C09144=1176.227,126.647,-53.704,-178.669,6.349,148.760
C09145=1176.232,126.397,-53.684,-178.672,6.347,148.760
C09146=1176.237,126.148,-53.664,-178.674,6.346,148.761
C09147=1176.242,125.899,-53.644,-178.677,6.344,148.761
C09148=1176.246,125.650,-53.625,-178.680,6.343,148.762
C09149=1176.251,125.401,-53.606,-178.683,6.341,148.762
C09150=1176.255,125.151,-53.586,-178.685,6.339,148.763
C09151=1176.260,124.903,-53.566,-178.688,6.338,148.763
C09152=1176.265,124.653,-53.546,-178.690,6.337,148.763
C09153=1176.270,124.404,-53.527,-178.693,6.335,148.764
C09154=1176.275,124.155,-53.507,-178.696,6.334,148.764
C09155=1176.280,123.906,-53.487,-178.698,6.333,148.765
C09156=1176.284,123.656,-53.467,-178.701,6.331,148.765
C09157=1176.290,123.407,-53.448,-178.704,6.330,148.766
C09158=1176.294,123.158,-53.429,-178.707,6.328,148.766
C09159=1176.299,122.909,-53.409,-178.709,6.327,148.767
C09160=1176.304,122.660,-53.390,-178.712,6.325,148.767
C09161=1176.308,122.411,-53.370,-178.715,6.324,148.768
C09162=1176.313,122.161,-53.350,-178.718,6.322,148.768
C09163=1176.318,121.912,-53.331,-178.720,6.321,148.768
C09164=1176.322,121.663,-53.312,-178.722,6.319,148.769
C09165=1176.327,121.414,-53.292,-178.726,6.318,148.769
C09166=1176.332,121.165,-53.273,-178.728,6.317,148.770
C09167=1176.337,120.915,-53.253,-178.730,6.315,148.770
C09168=1176.343,120.666,-53.234,-178.733,6.314,148.771
C09169=1176.347,120.417,-53.215,-178.736,6.312,148.771
C09170=1176.351,120.167,-53.195,-178.738,6.311,148.772
C09171=1176.357,119.919,-53.176,-178.741,6.310,148.772
C09172=1176.361,119.669,-53.156,-178.744,6.308,148.772
C09173=1176.366,119.420,-53.137,-178.747,6.306,148.773
C09174=1176.371,119.171,-53.118,-178.749,6.306,148.774
C09175=1176.375,118.921,-53.098,-178.752,6.304,148.774
C09176=1176.381,118.672,-53.079,-178.755,6.302,148.774
C09177=1176.385,118.423,-53.060,-178.757,6.302,148.775
C09178=1176.390,118.174,-53.041,-178.760,6.300,148.775
C09179=1176.395,117.925,-53.021,-178.763,6.298,148.776
C09180=1176.400,117.676,-53.002,-178.766,6.297,148.776
C09181=1176.404,117.427,-52.983,-178.768,6.296,148.777
C09182=1176.409,117.177,-52.963,-178.771,6.294,148.777
C09183=1176.414,116.928,-52.944,-178.773,6.292,148.778
C09184=1176.418,116.679,-52.925,-178.776,6.292,148.778
C09185=1176.424,116.430,-52.905,-178.779,6.290,148.779
C09186=1176.428,116.180,-52.886,-178.781,6.288,148.779
C09187=1176.433,115.931,-52.868,-178.783,6.287,148.779
C09188=1176.438,115.682,-52.848,-178.787,6.286,148.780
C09189=1176.443,115.433,-52.829,-178.789,6.284,148.780
C09190=1176.447,115.184,-52.810,-178.792,6.283,148.781
C09191=1176.453,114.935,-52.790,-178.795,6.282,148.782
C09192=1176.458,114.685,-52.771,-178.797,6.280,148.782
C09193=1176.462,114.436,-52.753,-178.800,6.278,148.782
C09194=1176.467,114.186,-52.733,-178.802,6.278,148.783
C09195=1176.473,113.938,-52.714,-178.805,6.276,148.783
C09196=1176.477,113.688,-52.695,-178.808,6.274,148.784
C09197=1176.482,113.439,-52.675,-178.810,6.274,148.784
C09198=1176.486,113.190,-52.657,-178.813,6.272,148.785
C09199=1176.492,112.941,-52.638,-178.816,6.270,148.785
C09200=1176.496,112.691,-52.619,-178.818,6.270,148.786
C09201=1176.501,112.443,-52.599,-178.822,6.268,148.786
C09202=1176.506,112.192,-52.580,-178.824,6.266,148.787
C09203=1176.511,111.944,-52.562,-178.826,6.266,148.787
C09204=1176.515,111.694,-52.542,-178.829,6.264,148.787
C09205=1176.520,111.445,-52.524,-178.832,6.262,148.788
C09206=1176.526,111.196,-52.505,-178.834,6.261,148.789
C09207=1176.530,110.947,-52.486,-178.837,6.260,148.789
C09208=1176.535,110.697,-52.467,-178.840,6.258,148.790
C09209=1176.539,110.448,-52.448,-178.842,6.257,148.790
C09210=1176.545,110.199,-52.429,-178.845,6.256,148.790
C09211=1176.549,109.949,-52.410,-178.848,6.254,148.791
C09212=1176.554,109.701,-52.391,-178.850,6.253,148.791
C09213=1176.559,109.451,-52.373,-178.853,6.252,148.792
C09214=1176.564,109.202,-52.354,-178.856,6.250,148.792
C09215=1176.568,108.953,-52.335,-178.859,6.249,148.793
C09216=1176.574,108.703,-52.316,-178.861,6.248,148.793
C09217=1176.578,108.455,-52.297,-178.864,6.246,148.794
C09218=1176.584,108.205,-52.279,-178.867,6.245,148.794
C09219=1176.588,107.956,-52.260,-178.869,6.244,148.795
C09220=1176.593,107.707,-52.242,-178.872,6.242,148.795
C09221=1176.597,107.457,-52.222,-178.875,6.241,148.796
C09222=1176.602,107.208,-52.204,-178.877,6.240,148.796
C09223=1176.608,106.959,-52.185,-178.880,6.239,148.797
C09224=1176.612,106.690,-52.165,-178.883,6.237,148.797
C09225=1176.618,106.422,-52.144,-178.886,6.236,148.798
C09226=1176.623,106.154,-52.125,-178.889,6.234,148.798
C09227=1176.628,105.885,-52.104,-178.892,6.233,148.799
C09228=1176.633,105.636,-52.086,-178.894,6.232,148.799
C09229=1176.638,105.387,-52.067,-178.897,6.230,148.800
C09230=1176.642,105.137,-52.048,-178.900,6.229,148.800
C09231=1176.647,104.888,-52.030,-178.902,6.228,148.801
C09232=1176.653,104.639,-52.011,-178.905,6.226,148.801
C09233=1176.657,104.389,-51.992,-178.908,6.225,148.802
C09234=1176.662,104.140,-51.974,-178.910,6.224,148.802
C09235=1176.667,103.891,-51.955,-178.913,6.222,148.803
C09236=1176.671,103.641,-51.937,-178.915,6.222,148.803
C09237=1176.676,103.392,-51.919,-178.918,6.220,148.804
C09238=1176.682,103.143,-51.900,-178.921,6.218,148.804
C09239=1176.687,102.894,-51.882,-178.923,6.218,148.805
C09240=1176.691,102.644,-51.863,-178.926,6.216,148.805
C09241=1176.695,102.396,-51.845,-178.928,6.215,148.806
C09242=1176.701,102.146,-51.826,-178.931,6.214,148.806
C09243=1176.705,101.896,-51.808,-178.934,6.212,148.807
C09244=1176.710,101.648,-51.789,-178.937,6.212,148.807
C09245=1176.716,101.398,-51.770,-178.939,6.210,148.808
C09246=1176.721,101.149,-51.752,-178.942,6.209,148.808
C09247=1176.725,100.899,-51.734,-178.945,6.208,148.809
C09248=1176.730,100.651,-51.715,-178.947,6.206,148.809
C09249=1176.735,100.401,-51.697,-178.950,6.205,148.810
C09250=1176.740,100.152,-51.679,-178.953,6.204,148.810
C09251=1176.744,99.902,-51.660,-178.955,6.203,148.811
C09252=1176.749,99.654,-51.642,-178.958,6.201,148.811
C09253=1176.754,99.405,-51.624,-178.961,6.200,148.812
C09254=1176.760,99.155,-51.605,-178.963,6.199,148.812
C09255=1176.764,98.905,-51.587,-178.966,6.197,148.813
C09256=1176.769,98.656,-51.569,-178.968,6.196,148.813
C09257=1176.773,98.407,-51.550,-178.971,6.195,148.814
C09258=1176.778,98.158,-51.532,-178.974,6.193,148.814
C09259=1176.783,97.909,-51.514,-178.976,6.192,148.815
C09260=1176.788,97.659,-51.495,-178.979,6.191,148.815
C09261=1176.793,97.410,-51.477,-178.982,6.190,148.816
C09262=1176.798,97.161,-51.459,-178.984,6.188,148.816
C09263=1176.803,96.911,-51.441,-178.987,6.188,148.817
C09264=1176.808,96.662,-51.423,-178.990,6.186,148.817
C09265=1176.812,96.412,-51.405,-178.992,6.184,148.818
C09266=1176.817,96.164,-51.386,-178.995,6.184,148.818
C09267=1176.822,95.915,-51.368,-178.998,6.182,148.819
C09268=1176.827,95.665,-51.350,-179.000,6.182,148.819
C09269=1176.832,95.416,-51.332,-179.003,6.180,148.820
C09270=1176.837,95.167,-51.314,-179.005,6.179,148.820
C09271=1176.842,94.917,-51.295,-179.008,6.178,148.821
C09272=1176.846,94.668,-51.277,-179.011,6.177,148.821
C09273=1176.851,94.419,-51.259,-179.014,6.175,148.822
C09274=1176.856,94.169,-51.241,-179.017,6.174,148.822
C09275=1176.861,93.920,-51.224,-179.019,6.173,148.823
C09276=1176.866,93.671,-51.206,-179.022,6.171,148.823
C09277=1176.871,93.422,-51.188,-179.024,6.171,148.824
C09278=1176.875,93.172,-51.169,-179.027,6.169,148.824
C09279=1176.880,92.923,-51.151,-179.029,6.168,148.825
C09280=1176.885,92.673,-51.134,-179.032,6.167,148.825
C09281=1176.890,92.424,-51.116,-179.035,6.166,148.826
C09282=1176.895,92.175,-51.098,-179.037,6.164,148.826
C09283=1176.900,91.925,-51.080,-179.041,6.163,148.827
C09284=1176.905,91.676,-51.062,-179.043,6.162,148.827
C09285=1176.910,91.427,-51.044,-179.045,6.160,148.828
C09286=1176.915,91.178,-51.026,-179.048,6.160,148.828
C09287=1176.920,90.929,-51.008,-179.051,6.158,148.829
C09288=1176.924,90.679,-50.990,-179.053,6.158,148.829
C09289=1176.929,90.429,-50.972,-179.056,6.156,148.830
C09290=1176.934,90.180,-50.955,-179.058,6.155,148.830
C09291=1176.939,89.931,-50.937,-179.062,6.154,148.831
C09292=1176.944,89.682,-50.919,-179.064,6.153,148.831
C09293=1176.949,89.432,-50.901,-179.067,6.151,148.832
C09294=1176.954,89.183,-50.883,-179.069,6.150,148.832
C09295=1176.959,88.933,-50.865,-179.072,6.149,148.833
C09296=1176.963,88.685,-50.848,-179.074,6.148,148.833
C09297=1176.968,88.435,-50.830,-179.077,6.146,148.834
C09298=1176.973,88.186,-50.812,-179.080,6.146,148.835
C09299=1176.978,87.936,-50.795,-179.082,6.144,148.835
C09300=1176.983,87.687,-50.777,-179.085,6.144,148.836
C09301=1176.988,87.438,-50.759,-179.088,6.142,148.836
C09302=1176.993,87.188,-50.741,-179.090,6.141,148.837
C09303=1176.998,86.939,-50.724,-179.093,6.140,148.837
C09304=1177.003,86.690,-50.706,-179.095,6.139,148.838
C09305=1177.007,86.441,-50.688,-179.098,6.137,148.838
C09306=1177.013,86.191,-50.671,-179.101,6.137,148.839
C09307=1177.018,85.942,-50.653,-179.104,6.135,148.839
C09308=1177.022,85.693,-50.635,-179.106,6.134,148.840
C09309=1177.028,85.443,-50.618,-179.109,6.133,148.840
C09310=1177.032,85.194,-50.600,-179.111,6.132,148.841
C09311=1177.037,84.944,-50.583,-179.114,6.130,148.841
C09312=1177.042,84.695,-50.565,-179.117,6.130,148.842
C09313=1177.047,84.446,-50.547,-179.119,6.128,148.842
C09314=1177.052,84.196,-50.530,-179.122,6.128,148.843
C09315=1177.056,83.947,-50.512,-179.125,6.126,148.843
C09316=1177.061,83.698,-50.495,-179.127,6.125,148.844
C09317=1177.066,83.448,-50.477,-179.130,6.124,148.844
C09318=1177.071,83.199,-50.459,-179.133,6.123,148.845
C09319=1177.077,82.949,-50.442,-179.135,6.121,148.845
C09320=1177.081,82.701,-50.425,-179.138,6.120,148.846
C09321=1177.086,82.451,-50.407,-179.141,6.119,148.847
C09322=1177.091,82.202,-50.389,-179.143,6.118,148.847
C09323=1177.095,81.952,-50.373,-179.146,6.117,148.848
C09324=1177.100,81.703,-50.355,-179.148,6.116,148.848
C09325=1177.106,81.454,-50.338,-179.151,6.115,148.849
C09326=1177.111,81.205,-50.320,-179.154,6.114,148.849
C09327=1177.115,80.955,-50.303,-179.157,6.112,148.850
C09328=1177.120,80.687,-50.284,-179.159,6.111,148.850
C09329=1177.126,80.418,-50.265,-179.162,6.110,148.851
C09330=1177.132,80.150,-50.247,-179.165,6.109,148.852
C09331=1177.137,79.881,-50.229,-179.167,6.108,148.852
C09332=1177.141,79.632,-50.211,-179.171,6.107,148.853
C09333=1177.147,79.382,-50.193,-179.173,6.106,148.853
C09334=1177.151,79.134,-50.176,-179.176,6.104,148.854
C09335=1177.156,78.884,-50.159,-179.178,6.103,148.854
C09336=1177.161,78.634,-50.141,-179.181,6.103,148.855
C09337=1177.166,78.386,-50.124,-179.184,6.101,148.855
C09338=1177.171,78.136,-50.107,-179.186,6.101,148.856
C09339=1177.175,77.887,-50.090,-179.189,6.099,148.856
C09340=1177.181,77.637,-50.072,-179.191,6.098,148.857
C09341=1177.186,77.388,-50.055,-179.194,6.097,148.857
C09342=1177.190,77.139,-50.038,-179.196,6.096,148.858
C09343=1177.195,76.889,-50.021,-179.200,6.094,148.858
C09344=1177.200,76.640,-50.004,-179.202,6.094,148.859
C09345=1177.205,76.391,-49.986,-179.204,6.093,148.860
C09346=1177.210,76.141,-49.969,-179.207,6.091,148.860
C09347=1177.215,75.892,-49.952,-179.210,6.091,148.861
C09348=1177.220,75.642,-49.935,-179.212,6.089,148.861
C09349=1177.225,75.394,-49.918,-179.215,6.089,148.862
C09350=1177.230,75.144,-49.901,-179.218,6.087,148.862
C09351=1177.235,74.894,-49.884,-179.220,6.086,148.863
C09352=1177.240,74.645,-49.867,-179.223,6.085,148.863
C09353=1177.244,74.396,-49.849,-179.226,6.084,148.864
C09354=1177.250,74.147,-49.833,-179.228,6.083,148.864
C09355=1177.254,73.897,-49.816,-179.231,6.082,148.865
C09356=1177.260,73.647,-49.799,-179.233,6.081,148.865
C09357=1177.264,73.398,-49.782,-179.237,6.080,148.866
C09358=1177.269,73.149,-49.764,-179.239,6.079,148.866
C09359=1177.274,72.900,-49.748,-179.241,6.078,148.867
C09360=1177.279,72.650,-49.730,-179.244,6.077,148.868
C09361=1177.284,72.401,-49.714,-179.247,6.076,148.868
C09362=1177.289,72.151,-49.696,-179.249,6.074,148.869
C09363=1177.294,71.902,-49.680,-179.252,6.074,148.869
C09364=1177.299,71.652,-49.663,-179.255,6.072,148.870
C09365=1177.304,71.403,-49.646,-179.257,6.072,148.870
C09366=1177.309,71.154,-49.628,-179.260,6.071,148.871
C09367=1177.314,70.905,-49.612,-179.263,6.069,148.871
C09368=1177.319,70.655,-49.595,-179.265,6.068,148.872
C09369=1177.323,70.406,-49.578,-179.268,6.067,148.873
C09370=1177.328,70.156,-49.561,-179.270,6.066,148.873
C09371=1177.334,69.907,-49.544,-179.273,6.066,148.874
C09372=1177.338,69.657,-49.528,-179.276,6.064,148.874
C09373=1177.343,69.408,-49.511,-179.278,6.063,148.875
C09374=1177.348,69.159,-49.494,-179.281,6.062,148.875
C09375=1177.353,68.909,-49.478,-179.284,6.061,148.876
C09376=1177.358,68.660,-49.460,-179.286,6.060,148.876
C09377=1177.363,68.410,-49.444,-179.289,6.059,148.877
C09378=1177.368,68.161,-49.427,-179.291,6.058,148.877
C09379=1177.373,67.912,-49.410,-179.294,6.058,148.878
C09380=1177.377,67.662,-49.393,-179.296,6.056,148.878
C09381=1177.383,67.413,-49.377,-179.299,6.055,148.879
C09382=1177.388,67.163,-49.360,-179.302,6.054,148.880
C09383=1177.392,66.914,-49.343,-179.304,6.053,148.880
C09384=1177.397,66.665,-49.327,-179.307,6.052,148.881
C09385=1177.403,66.415,-49.310,-179.310,6.051,148.881
C09386=1177.407,66.166,-49.293,-179.312,6.050,148.882
C09387=1177.412,65.917,-49.277,-179.315,6.050,148.882
C09388=1177.418,65.667,-49.260,-179.317,6.048,148.883
C09389=1177.422,65.417,-49.243,-179.320,6.047,148.883
C09390=1177.427,65.168,-49.227,-179.323,6.046,148.884
C09391=1177.432,64.919,-49.210,-179.325,6.045,148.885
C09392=1177.437,64.669,-49.193,-179.327,6.044,148.885
C09393=1177.442,64.420,-49.177,-179.331,6.043,148.886
C09394=1177.446,64.171,-49.160,-179.333,6.042,148.886
C09395=1177.452,63.922,-49.145,-179.335,6.042,148.887
C09396=1177.457,63.672,-49.127,-179.339,6.040,148.887
C09397=1177.462,63.422,-49.111,-179.341,6.039,148.888
C09398=1177.467,63.173,-49.094,-179.343,6.039,148.888
C09399=1177.471,62.924,-49.078,-179.346,6.037,148.889
C09400=1177.477,62.674,-49.062,-179.349,6.037,148.890
C09401=1177.482,62.425,-49.045,-179.352,6.035,148.890
C09402=1177.486,62.175,-49.028,-179.354,6.034,148.891
C09403=1177.491,61.927,-49.012,-179.356,6.033,148.891
C09404=1177.496,61.676,-48.996,-179.360,6.032,148.892
C09405=1177.502,61.427,-48.979,-179.362,6.031,148.892
C09406=1177.506,61.178,-48.962,-179.364,6.031,148.893
C09407=1177.511,60.929,-48.946,-179.367,6.029,148.893
C09408=1177.516,60.679,-48.930,-179.370,6.029,148.894
C09409=1177.521,60.429,-48.913,-179.372,6.028,148.895
C09410=1177.526,60.181,-48.897,-179.375,6.026,148.895
C09411=1177.531,59.930,-48.881,-179.378,6.026,148.896
C09412=1177.536,59.681,-48.864,-179.380,6.025,148.896
C09413=1177.541,59.432,-48.848,-179.383,6.024,148.897
C09414=1177.546,59.183,-48.832,-179.385,6.023,148.897
C09415=1177.551,58.933,-48.815,-179.388,6.022,148.898
C09416=1177.556,58.684,-48.799,-179.391,6.021,148.898
C09417=1177.561,58.434,-48.783,-179.393,6.020,148.899
C09418=1177.566,58.185,-48.767,-179.395,6.019,148.899
C09419=1177.571,57.935,-48.750,-179.399,6.018,148.900
C09420=1177.576,57.686,-48.734,-179.401,6.017,148.901
C09421=1177.581,57.437,-48.717,-179.403,6.016,148.901
C09422=1177.586,57.187,-48.702,-179.407,6.015,148.902
C09423=1177.591,56.938,-48.685,-179.409,6.014,148.902
C09424=1177.596,56.688,-48.669,-179.411,6.014,148.903
C09425=1177.600,56.439,-48.653,-179.414,6.013,148.903
C09426=1177.606,56.190,-48.637,-179.417,6.011,148.904
C09427=1177.610,55.940,-48.620,-179.419,6.011,148.905
C09428=1177.616,55.691,-48.605,-179.422,6.010,148.905
C09429=1177.620,55.441,-48.588,-179.425,6.009,148.906
C09430=1177.626,55.192,-48.573,-179.427,6.008,148.906
C09431=1177.630,54.942,-48.556,-179.430,6.007,148.907
C09432=1177.636,54.674,-48.539,-179.432,6.006,148.907
C09433=1177.641,54.405,-48.522,-179.435,6.005,148.908
C09434=1177.646,54.137,-48.504,-179.438,6.004,148.909
C09435=1177.651,53.868,-48.487,-179.441,6.003,148.909
C09436=1177.657,53.619,-48.471,-179.444,6.002,148.910
C09437=1177.661,53.369,-48.455,-179.446,6.001,148.911
C09438=1177.667,53.120,-48.439,-179.448,6.000,148.911
C09439=1177.671,52.870,-48.423,-179.451,6.000,148.912
C09440=1177.677,52.621,-48.407,-179.454,5.998,148.912
C09441=1177.682,52.372,-48.391,-179.456,5.998,148.913
C09442=1177.686,52.122,-48.374,-179.459,5.997,148.913
C09443=1177.692,51.873,-48.359,-179.462,5.995,148.914
C09444=1177.697,51.623,-48.343,-179.464,5.995,148.915
C09445=1177.702,51.374,-48.327,-179.466,5.994,148.915
C09446=1177.706,51.124,-48.311,-179.469,5.993,148.916
C09447=1177.712,50.875,-48.294,-179.472,5.992,148.916
C09448=1177.717,50.626,-48.279,-179.474,5.991,148.917
C09449=1177.722,50.376,-48.263,-179.477,5.991,148.917
C09450=1177.727,50.126,-48.247,-179.480,5.989,148.918
C09451=1177.731,49.877,-48.231,-179.483,5.989,148.919
C09452=1177.736,49.628,-48.216,-179.485,5.988,148.919
C09453=1177.742,49.378,-48.200,-179.487,5.987,148.920
C09454=1177.746,49.129,-48.183,-179.491,5.986,148.920
C09455=1177.751,48.879,-48.168,-179.493,5.985,148.921
C09456=1177.757,48.630,-48.152,-179.495,5.985,148.921
C09457=1177.762,48.380,-48.136,-179.497,5.984,148.922
C09458=1177.766,48.131,-48.120,-179.501,5.982,148.923
C09459=1177.771,47.882,-48.105,-179.503,5.981,148.923
C09460=1177.776,47.632,-48.089,-179.505,5.981,148.924
C09461=1177.782,47.382,-48.073,-179.508,5.980,148.924
C09462=1177.787,47.134,-48.057,-179.511,5.979,148.925
C09463=1177.791,46.884,-48.041,-179.514,5.978,148.925
C09464=1177.796,46.634,-48.026,-179.516,5.977,148.926
C09465=1177.801,46.385,-48.011,-179.518,5.977,148.927
C09466=1177.806,46.135,-47.995,-179.522,5.976,148.927
C09467=1177.812,45.886,-47.979,-179.524,5.975,148.928
C09468=1177.817,45.637,-47.963,-179.526,5.974,148.928
C09469=1177.821,45.387,-47.947,-179.528,5.973,148.929
C09470=1177.826,45.138,-47.932,-179.532,5.972,148.929
C09471=1177.831,44.888,-47.916,-179.534,5.971,148.930
C09472=1177.836,44.638,-47.900,-179.536,5.971,148.931
C09473=1177.841,44.389,-47.885,-179.539,5.970,148.931
C09474=1177.846,44.140,-47.870,-179.542,5.968,148.932
C09475=1177.852,43.890,-47.854,-179.545,5.968,148.932
C09476=1177.856,43.641,-47.837,-179.547,5.967,148.933
C09477=1177.861,43.392,-47.822,-179.549,5.967,148.933
C09478=1177.866,43.142,-47.807,-179.553,5.965,148.934
C09479=1177.871,42.892,-47.791,-179.555,5.964,148.935
C09480=1177.876,42.643,-47.776,-179.557,5.964,148.935
C09481=1177.881,42.394,-47.760,-179.559,5.963,148.936
C09482=1177.886,42.144,-47.745,-179.563,5.962,148.936
C09483=1177.891,41.894,-47.729,-179.565,5.961,148.937
C09484=1177.896,41.645,-47.714,-179.568,5.960,148.937
C09485=1177.901,41.396,-47.698,-179.570,5.960,148.938
C09486=1177.907,41.146,-47.683,-179.572,5.959,148.939
C09487=1177.911,40.897,-47.668,-179.576,5.958,148.939
C09488=1177.916,40.647,-47.652,-179.578,5.957,148.940
C09489=1177.921,40.398,-47.636,-179.580,5.956,148.940
C09490=1177.926,40.149,-47.621,-179.583,5.956,148.941
C09491=1177.931,39.899,-47.605,-179.586,5.954,148.941
C09492=1177.936,39.649,-47.590,-179.588,5.954,148.942
C09493=1177.941,39.400,-47.574,-179.591,5.953,148.943
C09494=1177.947,39.150,-47.560,-179.593,5.952,148.943
C09495=1177.951,38.901,-47.545,-179.596,5.952,148.944
C09496=1177.957,38.651,-47.529,-179.599,5.950,148.944
C09497=1177.961,38.401,-47.513,-179.601,5.950,148.945
C09498=1177.966,38.152,-47.498,-179.604,5.949,148.946
C09499=1177.971,37.903,-47.482,-179.606,5.948,148.946
C09500=1177.976,37.654,-47.467,-179.609,5.948,148.947
C09501=1177.982,37.404,-47.452,-179.612,5.946,148.948
C09502=1177.986,37.155,-47.438,-179.614,5.946,148.948
C09503=1177.991,36.904,-47.422,-179.617,5.945,148.949
C09504=1177.997,36.655,-47.406,-179.619,5.944,148.949
C09505=1178.001,36.406,-47.391,-179.621,5.944,148.950
C09506=1178.007,36.157,-47.375,-179.625,5.942,148.950
C09507=1178.011,35.908,-47.360,-179.627,5.941,148.951
C09508=1178.017,35.657,-47.346,-179.629,5.941,148.952
C09509=1178.022,35.408,-47.331,-179.632,5.940,148.952
C09510=1178.026,35.158,-47.315,-179.634,5.940,148.953
C09511=1178.031,34.909,-47.300,-179.638,5.938,148.953
C09512=1178.037,34.659,-47.285,-179.640,5.937,148.954
C09513=1178.041,34.410,-47.270,-179.642,5.937,148.954
C09514=1178.047,34.161,-47.254,-179.645,5.936,148.955
C09515=1178.051,33.912,-47.239,-179.647,5.936,148.956
C09516=1178.057,33.662,-47.224,-179.650,5.935,148.956
C09517=1178.062,33.412,-47.209,-179.653,5.933,148.957
C09518=1178.067,33.162,-47.193,-179.655,5.933,148.957
C09519=1178.071,32.913,-47.178,-179.658,5.932,148.958
C09520=1178.077,32.663,-47.164,-179.660,5.932,148.959
C09521=1178.082,32.414,-47.149,-179.663,5.931,148.959
C09522=1178.087,32.165,-47.133,-179.666,5.930,148.960
C09523=1178.092,31.915,-47.119,-179.668,5.929,148.960
C09524=1178.097,31.666,-47.104,-179.671,5.928,148.961
C09525=1178.102,31.417,-47.088,-179.673,5.928,148.961
C09526=1178.107,31.167,-47.074,-179.675,5.927,148.962
C09527=1178.112,30.917,-47.058,-179.678,5.927,148.963
C09528=1178.117,30.668,-47.044,-179.680,5.926,148.963
C09529=1178.123,30.418,-47.028,-179.683,5.924,148.964
C09530=1178.127,30.169,-47.013,-179.686,5.924,148.965
C09531=1178.132,29.919,-46.999,-179.688,5.923,148.965
C09532=1178.137,29.669,-46.983,-179.691,5.923,148.966
C09533=1178.142,29.420,-46.969,-179.693,5.922,148.966
C09534=1178.147,29.171,-46.954,-179.696,5.921,148.967
C09535=1178.152,28.921,-46.939,-179.699,5.920,148.968
C09536=1178.157,28.652,-46.923,-179.702,5.919,148.968
C09537=1178.163,28.383,-46.906,-179.704,5.919,148.969
C09538=1178.168,28.115,-46.891,-179.707,5.917,148.969
C09539=1178.174,27.845,-46.874,-179.710,5.917,148.970
C09540=1178.179,27.596,-46.860,-179.712,5.916,148.971
C09541=1178.184,27.347,-46.845,-179.714,5.915,148.971
C09542=1178.189,27.097,-46.830,-179.717,5.915,148.972
C09543=1178.194,26.848,-46.815,-179.720,5.914,148.973
C09544=1178.199,26.598,-46.801,-179.722,5.913,148.973
C09545=1178.204,26.349,-46.786,-179.725,5.912,148.974
C09546=1178.209,26.099,-46.771,-179.728,5.912,148.974
C09547=1178.214,25.850,-46.756,-179.730,5.911,148.975
C09548=1178.219,25.600,-46.742,-179.733,5.910,148.975
C09549=1178.224,25.350,-46.726,-179.735,5.910,148.976
C09550=1178.229,25.101,-46.712,-179.737,5.909,148.977
C09551=1178.234,24.852,-46.697,-179.740,5.909,148.977
C09552=1178.239,24.603,-46.683,-179.743,5.907,148.978
C09553=1178.245,24.353,-46.668,-179.745,5.906,148.978
C09554=1178.250,24.104,-46.653,-179.748,5.906,148.979
C09555=1178.255,23.854,-46.639,-179.750,5.905,148.980
C09556=1178.260,23.604,-46.625,-179.753,5.905,148.980
C09557=1178.265,23.355,-46.609,-179.756,5.904,148.981
C09558=1178.270,23.105,-46.595,-179.758,5.903,148.981
C09559=1178.275,22.856,-46.580,-179.760,5.903,148.982
C09560=1178.280,22.606,-46.565,-179.764,5.902,148.983
C09561=1178.285,22.357,-46.551,-179.766,5.901,148.983
C09562=1178.290,22.107,-46.536,-179.768,5.900,148.984
C09563=1178.295,21.857,-46.521,-179.771,5.899,148.984
C09564=1178.300,21.608,-46.507,-179.773,5.899,148.985
C09565=1178.305,21.358,-46.493,-179.776,5.898,148.986
C09566=1178.309,21.109,-46.478,-179.778,5.897,148.986
C09567=1178.315,20.859,-46.463,-179.781,5.897,148.987
C09568=1178.321,20.610,-46.449,-179.783,5.897,148.987
C09569=1178.325,20.361,-46.434,-179.786,5.895,148.988
C09570=1178.330,20.111,-46.420,-179.789,5.894,148.989
C09571=1178.335,19.861,-46.405,-179.791,5.894,148.989
C09572=1178.340,19.612,-46.391,-179.794,5.893,148.990
C09573=1178.345,19.362,-46.377,-179.796,5.893,148.990
C09574=1178.351,19.113,-46.361,-179.799,5.892,148.991
C09575=1178.356,18.863,-46.347,-179.801,5.891,148.992
C09576=1178.361,18.614,-46.333,-179.804,5.891,148.992
C09577=1178.366,18.364,-46.319,-179.806,5.890,148.993
C09578=1178.371,18.114,-46.305,-179.808,5.889,148.993
C09579=1178.376,17.865,-46.290,-179.811,5.889,148.994
C09580=1178.381,17.616,-46.275,-179.814,5.888,148.995
C09581=1178.386,17.366,-46.261,-179.817,5.887,148.995
C09582=1178.391,17.116,-46.247,-179.819,5.886,148.996
C09583=1178.396,16.867,-46.233,-179.821,5.885,148.996
C09584=1178.402,16.617,-46.218,-179.824,5.885,148.997
C09585=1178.406,16.368,-46.203,-179.827,5.884,148.998
C09586=1178.411,16.118,-46.189,-179.829,5.884,148.998
C09587=1178.416,15.869,-46.174,-179.831,5.883,148.999
C09588=1178.421,15.619,-46.160,-179.834,5.883,149.000
C09589=1178.427,15.370,-46.146,-179.836,5.882,149.000
C09590=1178.432,15.120,-46.132,-179.839,5.881,149.001
C09591=1178.437,14.870,-46.118,-179.842,5.881,149.001
C09592=1178.442,14.621,-46.103,-179.844,5.879,149.002
C09593=1178.447,14.371,-46.089,-179.847,5.879,149.002
C09594=1178.452,14.122,-46.075,-179.850,5.878,149.003
C09595=1178.457,13.872,-46.061,-179.852,5.877,149.004
C09596=1178.462,13.623,-46.047,-179.854,5.877,149.004
C09597=1178.467,13.373,-46.032,-179.857,5.876,149.005
C09598=1178.472,13.123,-46.018,-179.859,5.876,149.005
C09599=1178.478,12.874,-46.004,-179.862,5.875,149.006
C09600=1178.483,12.624,-45.990,-179.865,5.875,149.007
C09601=1178.487,12.375,-45.976,-179.867,5.874,149.007
C09602=1178.492,12.125,-45.961,-179.869,5.873,149.008
C09603=1178.497,11.875,-45.947,-179.872,5.873,149.009
C09604=1178.503,11.626,-45.933,-179.874,5.872,149.009
C09605=1178.508,11.377,-45.919,-179.877,5.871,149.010
C09606=1178.513,11.127,-45.905,-179.879,5.871,149.010
C09607=1178.517,10.878,-45.891,-179.882,5.870,149.011
C09608=1178.523,10.629,-45.877,-179.884,5.870,149.012
C09609=1178.528,10.379,-45.863,-179.888,5.868,149.012
C09610=1178.533,10.129,-45.848,-179.890,5.868,149.013
C09611=1178.538,9.880,-45.834,-179.892,5.867,149.013
C09612=1178.543,9.630,-45.820,-179.895,5.867,149.014
C09613=1178.548,9.381,-45.806,-179.897,5.866,149.015
C09614=1178.553,9.130,-45.792,-179.900,5.865,149.015
C09615=1178.559,8.881,-45.778,-179.902,5.865,149.016
C09616=1178.564,8.632,-45.764,-179.905,5.864,149.016
C09617=1178.568,8.382,-45.751,-179.907,5.863,149.017
C09618=1178.574,8.133,-45.737,-179.910,5.863,149.018
C09619=1178.579,7.883,-45.722,-179.912,5.862,149.018
C09620=1178.583,7.634,-45.708,-179.915,5.862,149.019
C09621=1178.589,7.383,-45.694,-179.917,5.861,149.020
C09622=1178.594,7.134,-45.681,-179.920,5.860,149.020
C09623=1178.599,6.885,-45.666,-179.922,5.860,149.021
C09624=1178.603,6.635,-45.653,-179.925,5.859,149.021
C09625=1178.609,6.386,-45.639,-179.927,5.859,149.022
C09626=1178.614,6.136,-45.625,-179.930,5.858,149.023
C09627=1178.619,5.886,-45.611,-179.932,5.858,149.023
C09628=1178.625,5.637,-45.597,-179.935,5.857,149.024
C09629=1178.629,5.388,-45.583,-179.937,5.856,149.024
C09630=1178.634,5.138,-45.570,-179.940,5.856,149.025
C09631=1178.640,4.889,-45.556,-179.942,5.855,149.026
C09632=1178.645,4.639,-45.542,-179.945,5.855,149.026
C09633=1178.650,4.389,-45.527,-179.947,5.854,149.027
C09634=1178.655,4.140,-45.515,-179.949,5.853,149.027
C09635=1178.660,3.890,-45.500,-179.952,5.853,149.028
C09636=1178.665,3.640,-45.486,-179.955,5.852,149.029
C09637=1178.671,3.391,-45.473,-179.957,5.851,149.029
C09638=1178.675,3.141,-45.459,-179.960,5.851,149.030
C09639=1178.680,2.892,-45.445,-179.962,5.850,149.031
C09640=1178.686,2.623,-45.430,-179.965,5.849,149.031
C09641=1178.691,2.354,-45.415,-179.968,5.849,149.032
C09642=1178.697,2.084,-45.400,-179.970,5.848,149.032
C09643=1178.703,1.815,-45.386,-179.973,5.847,149.033
C09644=1178.707,1.565,-45.373,-179.976,5.847,149.034
C09645=1178.712,1.316,-45.358,-179.978,5.846,149.035
C09646=1178.718,1.066,-45.345,-179.980,5.846,149.035
C09647=1178.722,0.817,-45.332,-179.983,5.845,149.036
C09648=1178.728,0.568,-45.318,-179.986,5.845,149.036
C09649=1178.733,0.317,-45.304,-179.988,5.844,149.037
C09650=1178.737,0.068,-45.290,-179.991,5.843,149.037
C09651=1178.743,-0.182,-45.277,-179.993,5.843,149.038
C09652=1178.748,-0.431,-45.263,-179.995,5.842,149.039
C09653=1178.753,-0.680,-45.250,-179.998,5.842,149.039
C09654=1178.758,-0.930,-45.236,179.999,5.841,149.040
C09655=1178.764,-1.179,-45.222,179.997,5.840,149.040
C09656=1178.768,-1.430,-45.209,179.994,5.840,149.041
C09657=1178.773,-1.679,-45.195,179.992,5.839,149.042
C09658=1178.779,-1.929,-45.182,179.989,5.839,149.043
C09659=1178.783,-2.178,-45.168,179.987,5.838,149.043
C09660=1178.789,-2.428,-45.155,179.984,5.838,149.044
C09661=1178.794,-2.678,-45.141,179.982,5.837,149.044
C09662=1178.799,-2.927,-45.128,179.980,5.836,149.045
C09663=1178.804,-3.177,-45.114,179.977,5.836,149.046
C09664=1178.809,-3.426,-45.101,179.974,5.835,149.046
C09665=1178.814,-3.676,-45.087,179.972,5.835,149.047
C09666=1178.820,-3.925,-45.074,179.969,5.834,149.047
C09667=1178.825,-4.175,-45.061,179.967,5.834,149.048
C09668=1178.830,-4.424,-45.047,179.965,5.833,149.049
C09669=1178.835,-4.674,-45.034,179.962,5.832,149.049
C09670=1178.840,-4.923,-45.020,179.959,5.832,149.050
C09671=1178.845,-5.173,-45.007,179.957,5.831,149.050
C09672=1178.851,-5.423,-44.994,179.955,5.831,149.051
C09673=1178.855,-5.672,-44.980,179.952,5.831,149.052
C09674=1178.861,-5.922,-44.967,179.950,5.830,149.052
C09675=1178.866,-6.172,-44.953,179.948,5.830,149.053
C09676=1178.871,-6.421,-44.940,179.945,5.829,149.054
C09677=1178.876,-6.671,-44.926,179.943,5.828,149.054
C09678=1178.881,-6.920,-44.913,179.940,5.828,149.055
C09679=1178.886,-7.170,-44.899,179.937,5.827,149.055
C09680=1178.891,-7.420,-44.887,179.935,5.827,149.056
C09681=1178.896,-7.669,-44.873,179.933,5.826,149.057
C09682=1178.901,-7.919,-44.860,179.930,5.826,149.057
C09683=1178.907,-8.169,-44.846,179.927,5.825,149.058
C09684=1178.911,-8.418,-44.833,179.925,5.824,149.058
C09685=1178.917,-8.667,-44.821,179.922,5.824,149.059
C09686=1178.922,-8.917,-44.807,179.920,5.823,149.060
C09687=1178.927,-9.167,-44.794,179.918,5.823,149.060
C09688=1178.932,-9.416,-44.780,179.915,5.822,149.061
C09689=1178.937,-9.666,-44.767,179.912,5.822,149.062
C09690=1178.942,-9.916,-44.754,179.910,5.821,149.062
C09691=1178.947,-10.165,-44.741,179.907,5.820,149.063
C09692=1178.952,-10.415,-44.727,179.905,5.820,149.064
C09693=1178.958,-10.664,-44.714,179.903,5.820,149.064
C09694=1178.963,-10.914,-44.702,179.901,5.819,149.065
C09695=1178.968,-11.164,-44.688,179.898,5.819,149.065
C09696=1178.973,-11.413,-44.675,179.896,5.818,149.066
C09697=1178.978,-11.663,-44.661,179.893,5.818,149.067
C09698=1178.983,-11.912,-44.649,179.890,5.817,149.067
C09699=1178.988,-12.162,-44.636,179.888,5.817,149.068
C09700=1178.993,-12.412,-44.623,179.886,5.816,149.068
C09701=1178.998,-12.661,-44.609,179.883,5.815,149.069
C09702=1179.004,-12.910,-44.596,179.880,5.815,149.070
C09703=1179.009,-13.160,-44.583,179.878,5.814,149.070
C09704=1179.014,-13.410,-44.571,179.875,5.814,149.071
C09705=1179.019,-13.660,-44.557,179.873,5.813,149.072
C09706=1179.024,-13.909,-44.544,179.871,5.812,149.072
C09707=1179.029,-14.159,-44.532,179.869,5.813,149.073
C09708=1179.035,-14.409,-44.518,179.866,5.812,149.073
C09709=1179.039,-14.658,-44.505,179.864,5.811,149.074
C09710=1179.045,-14.907,-44.492,179.861,5.811,149.075
C09711=1179.050,-15.157,-44.479,179.858,5.810,149.075
C09712=1179.055,-15.407,-44.466,179.856,5.810,149.076
C09713=1179.060,-15.656,-44.454,179.854,5.809,149.076
C09714=1179.065,-15.906,-44.440,179.851,5.809,149.077
C09715=1179.070,-16.156,-44.427,179.848,5.808,149.078
C09716=1179.076,-16.405,-44.415,179.846,5.807,149.078
C09717=1179.081,-16.655,-44.401,179.843,5.807,149.079
C09718=1179.086,-16.905,-44.389,179.841,5.807,149.080
C09719=1179.091,-17.154,-44.376,179.839,5.807,149.080
C09720=1179.096,-17.404,-44.363,179.836,5.806,149.081
C09721=1179.101,-17.654,-44.350,179.834,5.806,149.082
C09722=1179.107,-17.903,-44.337,179.832,5.805,149.082
C09723=1179.111,-18.153,-44.324,179.829,5.804,149.083
C09724=1179.116,-18.402,-44.312,179.826,5.804,149.083
C09725=1179.122,-18.652,-44.299,179.824,5.803,149.084
C09726=1179.127,-18.901,-44.286,179.821,5.803,149.085
C09727=1179.132,-19.151,-44.273,179.819,5.802,149.085
C09728=1179.137,-19.401,-44.260,179.817,5.802,149.086
C09729=1179.143,-19.650,-44.247,179.815,5.802,149.086
C09730=1179.147,-19.900,-44.234,179.812,5.801,149.087
C09731=1179.152,-20.149,-44.222,179.809,5.801,149.088
C09732=1179.157,-20.399,-44.209,179.807,5.800,149.088
C09733=1179.163,-20.648,-44.196,179.804,5.799,149.089
C09734=1179.168,-20.899,-44.184,179.802,5.799,149.090
C09735=1179.173,-21.148,-44.171,179.800,5.798,149.090
C09736=1179.178,-21.398,-44.158,179.797,5.798,149.091
C09737=1179.184,-21.647,-44.146,179.795,5.798,149.092
C09738=1179.188,-21.897,-44.133,179.793,5.797,149.092
C09739=1179.194,-22.147,-44.120,179.790,5.797,149.093
C09740=1179.199,-22.396,-44.107,179.787,5.796,149.093
C09741=1179.204,-22.646,-44.095,179.785,5.796,149.094
C09742=1179.209,-22.896,-44.082,179.783,5.795,149.095
C09743=1179.214,-23.145,-44.070,179.780,5.795,149.095
C09744=1179.220,-23.415,-44.056,179.777,5.794,149.096
C09745=1179.225,-23.684,-44.042,179.775,5.794,149.097
C09746=1179.230,-23.954,-44.028,179.772,5.793,149.097
C09747=1179.237,-24.224,-44.015,179.770,5.792,149.098
C09748=1179.242,-24.474,-44.002,179.767,5.792,149.099
C09749=1179.247,-24.723,-43.989,179.764,5.792,149.099
C09750=1179.252,-24.973,-43.977,179.763,5.792,149.100
C09751=1179.257,-25.223,-43.965,179.760,5.791,149.100
C09752=1179.262,-25.472,-43.952,179.757,5.791,149.101
C09753=1179.267,-25.722,-43.939,179.755,5.790,149.102
C09754=1179.272,-25.971,-43.927,179.753,5.789,149.102
C09755=1179.278,-26.222,-43.914,179.750,5.789,149.103
C09756=1179.283,-26.471,-43.902,179.747,5.788,149.104
C09757=1179.288,-26.720,-43.889,179.746,5.788,149.104
C09758=1179.294,-26.969,-43.877,179.743,5.788,149.105
C09759=1179.298,-27.220,-43.864,179.740,5.788,149.106
C09760=1179.304,-27.469,-43.852,179.738,5.787,149.106
C09761=1179.309,-27.719,-43.839,179.736,5.786,149.107
C09762=1179.314,-27.969,-43.827,179.733,5.786,149.107
C09763=1179.319,-28.218,-43.815,179.731,5.785,149.108
C09764=1179.324,-28.467,-43.802,179.729,5.785,149.109
C09765=1179.329,-28.718,-43.790,179.726,5.785,149.109
C09766=1179.334,-28.967,-43.777,179.724,5.784,149.110
C09767=1179.339,-29.217,-43.765,179.721,5.784,149.110
C09768=1179.345,-29.467,-43.753,179.718,5.783,149.111
C09769=1179.350,-29.716,-43.740,179.716,5.782,149.112
C09770=1179.355,-29.965,-43.727,179.714,5.782,149.112
C09771=1179.361,-30.215,-43.716,179.712,5.782,149.113
C09772=1179.365,-30.465,-43.703,179.709,5.782,149.114
C09773=1179.371,-30.715,-43.691,179.707,5.781,149.114
C09774=1179.376,-30.964,-43.678,179.704,5.781,149.115
C09775=1179.381,-31.214,-43.666,179.701,5.780,149.116
C09776=1179.386,-31.464,-43.654,179.699,5.779,149.116
C09777=1179.391,-31.713,-43.641,179.697,5.780,149.117
C09778=1179.397,-31.963,-43.629,179.694,5.779,149.117
C09779=1179.402,-32.212,-43.617,179.692,5.778,149.118
C09780=1179.407,-32.462,-43.605,179.690,5.778,149.119
C09781=1179.412,-32.711,-43.592,179.687,5.778,149.119
C09782=1179.418,-32.961,-43.580,179.685,5.777,149.120
C09783=1179.422,-33.211,-43.568,179.683,5.777,149.120
C09784=1179.427,-33.461,-43.556,179.680,5.777,149.121
C09785=1179.432,-33.710,-43.543,179.678,5.776,149.122
C09786=1179.438,-33.960,-43.531,179.675,5.775,149.122
C09787=1179.443,-34.210,-43.519,179.673,5.775,149.123
C09788=1179.448,-34.460,-43.507,179.671,5.775,149.123
C09789=1179.453,-34.709,-43.494,179.668,5.774,149.124
C09790=1179.459,-34.959,-43.482,179.666,5.774,149.125
C09791=1179.464,-35.208,-43.470,179.663,5.774,149.126
C09792=1179.469,-35.458,-43.458,179.661,5.773,149.126
C09793=1179.474,-35.707,-43.446,179.658,5.772,149.127
C09794=1179.479,-35.957,-43.434,179.656,5.773,149.127
C09795=1179.485,-36.207,-43.422,179.654,5.772,149.128
C09796=1179.490,-36.456,-43.410,179.651,5.771,149.129
C09797=1179.495,-36.706,-43.398,179.649,5.771,149.129
C09798=1179.500,-36.955,-43.385,179.646,5.770,149.130
C09799=1179.506,-37.205,-43.373,179.644,5.771,149.131
C09800=1179.510,-37.455,-43.362,179.642,5.770,149.131
C09801=1179.515,-37.704,-43.349,179.639,5.769,149.132
C09802=1179.521,-37.954,-43.337,179.637,5.769,149.132
C09803=1179.526,-38.204,-43.325,179.634,5.768,149.133
C09804=1179.531,-38.454,-43.313,179.633,5.768,149.134
C09805=1179.536,-38.703,-43.302,179.630,5.768,149.134
C09806=1179.541,-38.952,-43.289,179.627,5.768,149.135
C09807=1179.547,-39.202,-43.277,179.625,5.767,149.135
C09808=1179.552,-39.452,-43.265,179.622,5.766,149.136
C09809=1179.557,-39.702,-43.253,179.620,5.767,149.137
C09810=1179.562,-39.951,-43.241,179.618,5.766,149.137
C09811=1179.567,-40.201,-43.230,179.615,5.765,149.138
C09812=1179.573,-40.451,-43.218,179.613,5.765,149.139
C09813=1179.578,-40.701,-43.205,179.611,5.764,149.139
C09814=1179.583,-40.950,-43.194,179.609,5.764,149.140
C09815=1179.588,-41.200,-43.182,179.606,5.764,149.141
C09816=1179.593,-41.449,-43.169,179.603,5.764,149.141
C09817=1179.599,-41.699,-43.157,179.601,5.763,149.142
C09818=1179.603,-41.949,-43.146,179.598,5.762,149.142
C09819=1179.609,-42.199,-43.134,179.596,5.763,149.143
C09820=1179.614,-42.448,-43.122,179.594,5.762,149.144
C09821=1179.619,-42.698,-43.110,179.591,5.761,149.144
C09822=1179.624,-42.948,-43.098,179.589,5.761,149.145
C09823=1179.629,-43.198,-43.087,179.587,5.760,149.146
C09824=1179.635,-43.447,-43.075,179.585,5.761,149.146
C09825=1179.640,-43.696,-43.063,179.582,5.760,149.147
C09826=1179.645,-43.946,-43.051,179.580,5.759,149.147
C09827=1179.651,-44.196,-43.039,179.577,5.759,149.148
C09828=1179.655,-44.445,-43.028,179.575,5.759,149.149
C09829=1179.661,-44.695,-43.016,179.573,5.758,149.149
C09830=1179.666,-44.945,-43.003,179.570,5.758,149.150
C09831=1179.671,-45.194,-42.992,179.567,5.758,149.151
C09832=1179.676,-45.444,-42.980,179.565,5.757,149.151
C09833=1179.681,-45.694,-42.968,179.563,5.757,149.152
C09834=1179.686,-45.944,-42.957,179.561,5.757,149.153
C09835=1179.692,-46.193,-42.946,179.558,5.756,149.153
C09836=1179.698,-46.443,-42.934,179.556,5.755,149.154
C09837=1179.702,-46.693,-42.922,179.554,5.756,149.154
C09838=1179.707,-46.942,-42.910,179.551,5.755,149.155
C09839=1179.713,-47.192,-42.898,179.549,5.755,149.156
C09840=1179.718,-47.441,-42.887,179.546,5.754,149.156
C09841=1179.723,-47.691,-42.875,179.544,5.754,149.157
C09842=1179.728,-47.941,-42.863,179.542,5.754,149.157
C09843=1179.734,-48.190,-42.852,179.539,5.753,149.158
C09844=1179.739,-48.440,-42.840,179.537,5.752,149.159
C09845=1179.744,-48.690,-42.829,179.535,5.753,149.159
C09846=1179.749,-48.940,-42.817,179.532,5.752,149.160
C09847=1179.754,-49.189,-42.806,179.530,5.752,149.161
C09848=1179.760,-49.459,-42.793,179.527,5.751,149.161
C09849=1179.765,-49.730,-42.781,179.525,5.751,149.162
C09850=1179.771,-50.000,-42.768,179.522,5.750,149.163
C09851=1179.777,-50.270,-42.755,179.519,5.750,149.163
C09852=1179.782,-50.521,-42.744,179.517,5.750,149.164
C09853=1179.787,-50.770,-42.733,179.515,5.749,149.165
C09854=1179.793,-51.020,-42.721,179.512,5.749,149.165
C09855=1179.797,-51.270,-42.710,179.510,5.749,149.166
C09856=1179.803,-51.519,-42.698,179.508,5.749,149.166
C09857=1179.808,-51.769,-42.687,179.506,5.748,149.167
C09858=1179.813,-52.019,-42.675,179.503,5.748,149.168
C09859=1179.819,-52.269,-42.663,179.501,5.747,149.168
C09860=1179.823,-52.518,-42.652,179.499,5.747,149.169
C09861=1179.830,-52.767,-42.640,179.496,5.747,149.170
C09862=1179.834,-53.017,-42.629,179.494,5.746,149.170
C09863=1179.840,-53.267,-42.617,179.491,5.746,149.171
C09864=1179.844,-53.517,-42.606,179.489,5.746,149.171
C09865=1179.849,-53.766,-42.594,179.487,5.745,149.172
C09866=1179.855,-54.015,-42.583,179.484,5.745,149.173
C09867=1179.860,-54.265,-42.572,179.483,5.745,149.173
C09868=1179.865,-54.516,-42.560,179.480,5.744,149.174
C09869=1179.870,-54.765,-42.549,179.477,5.744,149.175
C09870=1179.876,-55.014,-42.538,179.475,5.743,149.175
C09871=1179.881,-55.264,-42.526,179.473,5.744,149.176
C09872=1179.886,-55.514,-42.514,179.470,5.743,149.177
C09873=1179.891,-55.764,-42.503,179.468,5.742,149.177
C09874=1179.896,-56.013,-42.492,179.465,5.742,149.178
C09875=1179.902,-56.263,-42.481,179.463,5.742,149.178
C09876=1179.907,-56.513,-42.470,179.461,5.741,149.179
C09877=1179.912,-56.763,-42.458,179.459,5.741,149.180
C09878=1179.917,-57.012,-42.447,179.456,5.741,149.180
C09879=1179.922,-57.261,-42.436,179.454,5.741,149.181
C09880=1179.928,-57.512,-42.425,179.452,5.740,149.181
C09881=1179.933,-57.761,-42.413,179.449,5.740,149.182
C09882=1179.939,-58.011,-42.402,179.447,5.740,149.183
C09883=1179.943,-58.260,-42.390,179.445,5.739,149.183
C09884=1179.948,-58.511,-42.380,179.442,5.739,149.184
C09885=1179.954,-58.761,-42.368,179.440,5.739,149.185
C09886=1179.959,-59.009,-42.357,179.438,5.738,149.185
C09887=1179.964,-59.259,-42.346,179.435,5.738,149.186
C09888=1179.969,-59.510,-42.335,179.433,5.737,149.186
C09889=1179.975,-59.759,-42.324,179.431,5.738,149.187
C09890=1179.980,-60.008,-42.312,179.428,5.737,149.188
C09891=1179.985,-60.258,-42.300,179.426,5.736,149.188
C09892=1179.990,-60.508,-42.290,179.424,5.737,149.189
C09893=1179.996,-60.758,-42.278,179.422,5.736,149.190
C09894=1180.001,-61.007,-42.267,179.419,5.736,149.190
C09895=1180.006,-61.257,-42.257,179.416,5.735,149.191
C09896=1180.011,-61.506,-42.246,179.415,5.735,149.191
C09897=1180.016,-61.756,-42.234,179.412,5.735,149.192
C09898=1180.021,-62.007,-42.223,179.409,5.734,149.193
C09899=1180.027,-62.255,-42.212,179.408,5.734,149.193
C09900=1180.032,-62.505,-42.200,179.405,5.734,149.194
C09901=1180.037,-62.756,-42.190,179.402,5.733,149.195
C09902=1180.042,-63.005,-42.179,179.401,5.733,149.195
C09903=1180.048,-63.255,-42.167,179.398,5.733,149.196
C09904=1180.053,-63.504,-42.157,179.396,5.733,149.197
C09905=1180.058,-63.754,-42.145,179.393,5.732,149.197
C09906=1180.063,-64.004,-42.135,179.391,5.732,149.198
C09907=1180.069,-64.253,-42.123,179.389,5.731,149.198
C09908=1180.074,-64.503,-42.112,179.386,5.731,149.199
C09909=1180.079,-64.753,-42.101,179.384,5.731,149.200
C09910=1180.084,-65.002,-42.091,179.382,5.730,149.200
C09911=1180.090,-65.253,-42.079,179.379,5.730,149.201
C09912=1180.095,-65.501,-42.068,179.377,5.730,149.202
C09913=1180.100,-65.752,-42.058,179.375,5.730,149.202
C09914=1180.105,-66.001,-42.047,179.373,5.729,149.203
C09915=1180.110,-66.251,-42.036,179.370,5.730,149.203
C09916=1180.116,-66.501,-42.025,179.368,5.729,149.204
C09917=1180.121,-66.751,-42.014,179.366,5.728,149.205
C09918=1180.126,-67.000,-42.003,179.364,5.728,149.205
C09919=1180.131,-67.250,-41.992,179.361,5.728,149.206
C09920=1180.137,-67.499,-41.981,179.359,5.728,149.207
C09921=1180.142,-67.750,-41.970,179.357,5.727,149.207
C09922=1180.147,-67.999,-41.959,179.354,5.727,149.208
C09923=1180.152,-68.249,-41.949,179.352,5.727,149.208
C09924=1180.157,-68.498,-41.938,179.350,5.726,149.209
C09925=1180.163,-68.748,-41.927,179.348,5.726,149.210
C09926=1180.168,-68.998,-41.915,179.345,5.726,149.210
C09927=1180.174,-69.247,-41.905,179.343,5.725,149.211
C09928=1180.178,-69.497,-41.894,179.341,5.725,149.211
C09929=1180.184,-69.747,-41.884,179.338,5.725,149.212
C09930=1180.189,-69.996,-41.872,179.336,5.724,149.213
C09931=1180.194,-70.246,-41.862,179.334,5.725,149.213
C09932=1180.199,-70.496,-41.852,179.331,5.724,149.214
C09933=1180.205,-70.746,-41.840,179.329,5.723,149.215
C09934=1180.210,-70.996,-41.830,179.327,5.724,149.215
C09935=1180.215,-71.245,-41.818,179.325,5.723,149.216
C09936=1180.221,-71.495,-41.808,179.322,5.723,149.216
C09937=1180.226,-71.745,-41.798,179.320,5.723,149.217
C09938=1180.231,-71.994,-41.787,179.318,5.722,149.218
C09939=1180.236,-72.244,-41.776,179.315,5.722,149.218
C09940=1180.241,-72.494,-41.766,179.313,5.722,149.219
C09941=1180.247,-72.744,-41.754,179.311,5.721,149.220
C09942=1180.253,-72.993,-41.744,179.308,5.721,149.220
C09943=1180.258,-73.243,-41.733,179.306,5.721,149.221
C09944=1180.263,-73.492,-41.722,179.304,5.721,149.221
C09945=1180.268,-73.743,-41.712,179.302,5.721,149.222
C09946=1180.273,-73.992,-41.701,179.299,5.720,149.223
C09947=1180.278,-74.242,-41.690,179.297,5.720,149.223
C09948=1180.284,-74.491,-41.680,179.295,5.720,149.224
C09949=1180.289,-74.742,-41.669,179.292,5.719,149.225
C09950=1180.294,-74.990,-41.658,179.290,5.719,149.225
C09951=1180.299,-75.241,-41.648,179.288,5.719,149.226
C09952=1180.306,-75.512,-41.637,179.286,5.719,149.226
C09953=1180.310,-75.782,-41.625,179.283,5.718,149.227
C09954=1180.316,-76.054,-41.613,179.280,5.718,149.228
C09955=1180.323,-76.324,-41.602,179.278,5.717,149.228
C09956=1180.328,-76.574,-41.591,179.276,5.717,149.229
C09957=1180.333,-76.824,-41.581,179.273,5.717,149.230
C09958=1180.338,-77.074,-41.570,179.272,5.717,149.230
C09959=1180.344,-77.324,-41.560,179.269,5.716,149.231
C09960=1180.348,-77.573,-41.549,179.267,5.716,149.231
C09961=1180.354,-77.823,-41.539,179.265,5.716,149.232
C09962=1180.360,-78.072,-41.528,179.262,5.716,149.233
C09963=1180.365,-78.323,-41.518,179.260,5.715,149.233
C09964=1180.370,-78.572,-41.508,179.258,5.715,149.234
C09965=1180.375,-78.822,-41.496,179.255,5.715,149.235
C09966=1180.380,-79.071,-41.486,179.253,5.714,149.235
C09967=1180.385,-79.322,-41.475,179.251,5.714,149.236
C09968=1180.390,-79.571,-41.466,179.249,5.714,149.236
C09969=1180.396,-79.820,-41.456,179.247,5.714,149.237
C09970=1180.401,-80.071,-41.445,179.244,5.714,149.238
C09971=1180.406,-80.320,-41.434,179.242,5.713,149.238
C09972=1180.411,-80.570,-41.424,179.240,5.713,149.239
C09973=1180.417,-80.819,-41.413,179.237,5.712,149.239
C09974=1180.422,-81.069,-41.403,179.235,5.712,149.240
C09975=1180.427,-81.319,-41.393,179.233,5.712,149.241
C09976=1180.433,-81.569,-41.382,179.231,5.712,149.241
C09977=1180.438,-81.819,-41.372,179.228,5.712,149.242
C09978=1180.444,-82.069,-41.362,179.226,5.711,149.243
C09979=1180.449,-82.318,-41.351,179.224,5.711,149.243
C09980=1180.453,-82.568,-41.341,179.222,5.711,149.244
C09981=1180.459,-82.817,-41.330,179.219,5.710,149.244
C09982=1180.464,-83.067,-41.320,179.217,5.710,149.245
C09983=1180.469,-83.317,-41.310,179.215,5.710,149.246
C09984=1180.475,-83.566,-41.299,179.212,5.710,149.246
C09985=1180.480,-83.816,-41.289,179.211,5.710,149.247
C09986=1180.486,-84.066,-41.279,179.208,5.709,149.248
C09987=1180.490,-84.315,-41.269,179.205,5.709,149.248
C09988=1180.495,-84.565,-41.259,179.204,5.709,149.249
C09989=1180.501,-84.815,-41.248,179.201,5.708,149.249
C09990=1180.507,-85.065,-41.238,179.200,5.708,149.250
C09991=1180.512,-85.315,-41.228,179.197,5.708,149.251
C09992=1180.517,-85.564,-41.217,179.194,5.708,149.251
C09993=1180.522,-85.814,-41.208,179.193,5.708,149.252
C09994=1180.527,-86.064,-41.197,179.190,5.707,149.253
C09995=1180.533,-86.313,-41.187,179.188,5.706,149.253
C09996=1180.538,-86.563,-41.177,179.186,5.707,149.254
//INST
///DATE 2021/06/15 17:25
///ATTR SC,RW,RJ
////FRAME ROBOT
///GROUP1 RB1
NOP
MOVL C00000 V=800.0 PL=0
MOVL C00001 V=800.0 PL=0
MOVL C00002 V=800.0 PL=0
MOVL C00003 V=800.0 PL=0
MOVL C00004 V=800.0 PL=0
MOVL C00005 V=800.0 PL=0
MOVL C00006 V=800.0 PL=0
MOVL C00007 V=800.0 PL=0
MOVL C00008 V=800.0 PL=0
MOVL C00009 V=800.0 PL=0
MOVL C00010 V=800.0 PL=0
MOVL C00011 V=800.0 PL=0
MOVL C00012 V=800.0 PL=0
MOVL C00013 V=800.0 PL=0
MOVL C00014 V=800.0 PL=0
MOVL C00015 V=800.0 PL=0
MOVL C00016 V=800.0 PL=0
MOVL C00017 V=800.0 PL=0
MOVL C00018 V=800.0 PL=0
MOVL C00019 V=800.0 PL=0
MOVL C00020 V=800.0 PL=0
MOVL C00021 V=800.0 PL=0
MOVL C00022 V=800.0 PL=0
MOVL C00023 V=800.0 PL=0
MOVL C00024 V=800.0 PL=0
MOVL C00025 V=800.0 PL=0
MOVL C00026 V=800.0 PL=0
MOVL C00027 V=800.0 PL=0
MOVL C00028 V=800.0 PL=0
MOVL C00029 V=800.0 PL=0
MOVL C00030 V=800.0 PL=0
MOVL C00031 V=800.0 PL=0
MOVL C00032 V=800.0 PL=0
MOVL C00033 V=800.0 PL=0
MOVL C00034 V=800.0 PL=0
MOVL C00035 V=800.0 PL=0
MOVL C00036 V=800.0 PL=0
MOVL C00037 V=800.0 PL=0
MOVL C00038 V=800.0 PL=0
MOVL C00039 V=800.0 PL=0
MOVL C00040 V=800.0 PL=0
MOVL C00041 V=800.0 PL=0
MOVL C00042 V=800.0 PL=0
MOVL C00043 V=800.0 PL=0
MOVL C00044 V=800.0 PL=0
MOVL C00045 V=800.0 PL=0
MOVL C00046 V=800.0 PL=0
MOVL C00047 V=800.0 PL=0
MOVL C00048 V=800.0 PL=0
MOVL C00049 V=800.0 PL=0
MOVL C00050 V=800.0 PL=0
MOVL C00051 V=800.0 PL=0
MOVL C00052 V=800.0 PL=0
MOVL C00053 V=800.0 PL=0
MOVL C00054 V=800.0 PL=0
MOVL C00055 V=800.0 PL=0
MOVL C00056 V=800.0 PL=0
MOVL C00057 V=800.0 PL=0
MOVL C00058 V=800.0 PL=0
MOVL C00059 V=800.0 PL=0
MOVL C00060 V=800.0 PL=0
MOVL C00061 V=800.0 PL=0
MOVL C00062 V=800.0 PL=0
MOVL C00063 V=800.0 PL=0
MOVL C00064 V=800.0 PL=0
MOVL C00065 V=800.0 PL=0
MOVL C00066 V=800.0 PL=0
MOVL C00067 V=800.0 PL=0
MOVL C00068 V=800.0 PL=0
MOVL C00069 V=800.0 PL=0
MOVL C00070 V=800.0 PL=0
MOVL C00071 V=800.0 PL=0
MOVL C00072 V=800.0 PL=0
MOVL C00073 V=800.0 PL=0
MOVL C00074 V=800.0 PL=0
MOVL C00075 V=800.0 PL=0
MOVL C00076 V=800.0 PL=0
MOVL C00077 V=800.0 PL=0
MOVL C00078 V=800.0 PL=0
MOVL C00079 V=800.0 PL=0
MOVL C00080 V=800.0 PL=0
MOVL C00081 V=800.0 PL=0
MOVL C00082 V=800.0 PL=0
MOVL C00083 V=800.0 PL=0
MOVL C00084 V=800.0 PL=0
MOVL C00085 V=800.0 PL=0
MOVL C00086 V=800.0 PL=0
MOVL C00087 V=800.0 PL=0
MOVL C00088 V=800.0 PL=0
MOVL C00089 V=800.0 PL=0
MOVL C00090 V=800.0 PL=0
MOVL C00091 V=800.0 PL=0
MOVL C00092 V=800.0 PL=0
MOVL C00093 V=800.0 PL=0
MOVL C00094 V=800.0 PL=0
MOVL C00095 V=800.0 PL=0
MOVL C00096 V=800.0 PL=0
MOVL C00097 V=800.0 PL=0
MOVL C00098 V=800.0 PL=0
MOVL C00099 V=800.0 PL=0
MOVL C00100 V=800.0 PL=0
MOVL C00101 V=800.0 PL=0
MOVL C00102 V=800.0 PL=0
MOVL C00103 V=800.0 PL=0
MOVL C00104 V=800.0 PL=0
MOVL C00105 V=800.0 PL=0
MOVL C00106 V=800.0 PL=0
MOVL C00107 V=800.0 PL=0
MOVL C00108 V=800.0 PL=0
MOVL C00109 V=800.0 PL=0
MOVL C00110 V=800.0 PL=0
MOVL C00111 V=800.0 PL=0
MOVL C00112 V=800.0 PL=0
MOVL C00113 V=800.0 PL=0
MOVL C00114 V=800.0 PL=0
MOVL C00115 V=800.0 PL=0
MOVL C00116 V=800.0 PL=0
MOVL C00117 V=800.0 PL=0
MOVL C00118 V=800.0 PL=0
MOVL C00119 V=800.0 PL=0
MOVL C00120 V=800.0 PL=0
MOVL C00121 V=800.0 PL=0
MOVL C00122 V=800.0 PL=0
MOVL C00123 V=800.0 PL=0
MOVL C00124 V=800.0 PL=0
MOVL C00125 V=800.0 PL=0
MOVL C00126 V=800.0 PL=0
MOVL C00127 V=800.0 PL=0
MOVL C00128 V=800.0 PL=0
MOVL C00129 V=800.0 PL=0
MOVL C00130 V=800.0 PL=0
MOVL C00131 V=800.0 PL=0
MOVL C00132 V=800.0 PL=0
MOVL C00133 V=800.0 PL=0
MOVL C00134 V=800.0 PL=0
MOVL C00135 V=800.0 PL=0
MOVL C00136 V=800.0 PL=0
MOVL C00137 V=800.0 PL=0
MOVL C00138 V=800.0 PL=0
MOVL C00139 V=800.0 PL=0
MOVL C00140 V=800.0 PL=0
MOVL C00141 V=800.0 PL=0
MOVL C00142 V=800.0 PL=0
MOVL C00143 V=800.0 PL=0
MOVL C00144 V=800.0 PL=0
MOVL C00145 V=800.0 PL=0
MOVL C00146 V=800.0 PL=0
MOVL C00147 V=800.0 PL=0
MOVL C00148 V=800.0 PL=0
MOVL C00149 V=800.0 PL=0
MOVL C00150 V=800.0 PL=0
MOVL C00151 V=800.0 PL=0
MOVL C00152 V=800.0 PL=0
MOVL C00153 V=800.0 PL=0
MOVL C00154 V=800.0 PL=0
MOVL C00155 V=800.0 PL=0
MOVL C00156 V=800.0 PL=0
MOVL C00157 V=800.0 PL=0
MOVL C00158 V=800.0 PL=0
MOVL C00159 V=800.0 PL=0
MOVL C00160 V=800.0 PL=0
MOVL C00161 V=800.0 PL=0
MOVL C00162 V=800.0 PL=0
MOVL C00163 V=800.0 PL=0
MOVL C00164 V=800.0 PL=0
MOVL C00165 V=800.0 PL=0
MOVL C00166 V=800.0 PL=0
MOVL C00167 V=800.0 PL=0
MOVL C00168 V=800.0 PL=0
MOVL C00169 V=800.0 PL=0
MOVL C00170 V=800.0 PL=0
MOVL C00171 V=800.0 PL=0
MOVL C00172 V=800.0 PL=0
MOVL C00173 V=800.0 PL=0
MOVL C00174 V=800.0 PL=0
MOVL C00175 V=800.0 PL=0
MOVL C00176 V=800.0 PL=0
MOVL C00177 V=800.0 PL=0
MOVL C00178 V=800.0 PL=0
MOVL C00179 V=800.0 PL=0
MOVL C00180 V=800.0 PL=0
MOVL C00181 V=800.0 PL=0
MOVL C00182 V=800.0 PL=0
MOVL C00183 V=800.0 PL=0
MOVL C00184 V=800.0 PL=0
MOVL C00185 V=800.0 PL=0
MOVL C00186 V=800.0 PL=0
MOVL C00187 V=800.0 PL=0
MOVL C00188 V=800.0 PL=0
MOVL C00189 V=800.0 PL=0
MOVL C00190 V=800.0 PL=0
MOVL C00191 V=800.0 PL=0
MOVL C00192 V=800.0 PL=0
MOVL C00193 V=800.0 PL=0
MOVL C00194 V=800.0 PL=0
MOVL C00195 V=800.0 PL=0
MOVL C00196 V=800.0 PL=0
MOVL C00197 V=800.0 PL=0
MOVL C00198 V=800.0 PL=0
MOVL C00199 V=800.0 PL=0
MOVL C00200 V=800.0 PL=0
MOVL C00201 V=800.0 PL=0
MOVL C00202 V=800.0 PL=0
MOVL C00203 V=800.0 PL=0
MOVL C00204 V=800.0 PL=0
MOVL C00205 V=800.0 PL=0
MOVL C00206 V=800.0 PL=0
MOVL C00207 V=800.0 PL=0
MOVL C00208 V=800.0 PL=0
MOVL C00209 V=800.0 PL=0
MOVL C00210 V=800.0 PL=0
MOVL C00211 V=800.0 PL=0
MOVL C00212 V=800.0 PL=0
MOVL C00213 V=800.0 PL=0
MOVL C00214 V=800.0 PL=0
MOVL C00215 V=800.0 PL=0
MOVL C00216 V=800.0 PL=0
MOVL C00217 V=800.0 PL=0
MOVL C00218 V=800.0 PL=0
MOVL C00219 V=800.0 PL=0
MOVL C00220 V=800.0 PL=0
MOVL C00221 V=800.0 PL=0
MOVL C00222 V=800.0 PL=0
MOVL C00223 V=800.0 PL=0
MOVL C00224 V=800.0 PL=0
MOVL C00225 V=800.0 PL=0
MOVL C00226 V=800.0 PL=0
MOVL C00227 V=800.0 PL=0
MOVL C00228 V=800.0 PL=0
MOVL C00229 V=800.0 PL=0
MOVL C00230 V=800.0 PL=0
MOVL C00231 V=800.0 PL=0
MOVL C00232 V=800.0 PL=0
MOVL C00233 V=800.0 PL=0
MOVL C00234 V=800.0 PL=0
MOVL C00235 V=800.0 PL=0
MOVL C00236 V=800.0 PL=0
MOVL C00237 V=800.0 PL=0
MOVL C00238 V=800.0 PL=0
MOVL C00239 V=800.0 PL=0
MOVL C00240 V=800.0 PL=0
MOVL C00241 V=800.0 PL=0
MOVL C00242 V=800.0 PL=0
MOVL C00243 V=800.0 PL=0
MOVL C00244 V=800.0 PL=0
MOVL C00245 V=800.0 PL=0
MOVL C00246 V=800.0 PL=0
MOVL C00247 V=800.0 PL=0
MOVL C00248 V=800.0 PL=0
MOVL C00249 V=800.0 PL=0
MOVL C00250 V=800.0 PL=0
MOVL C00251 V=800.0 PL=0
MOVL C00252 V=800.0 PL=0
MOVL C00253 V=800.0 PL=0
MOVL C00254 V=800.0 PL=0
MOVL C00255 V=800.0 PL=0
MOVL C00256 V=800.0 PL=0
MOVL C00257 V=800.0 PL=0
MOVL C00258 V=800.0 PL=0
MOVL C00259 V=800.0 PL=0
MOVL C00260 V=800.0 PL=0
MOVL C00261 V=800.0 PL=0
MOVL C00262 V=800.0 PL=0
MOVL C00263 V=800.0 PL=0
MOVL C00264 V=800.0 PL=0
MOVL C00265 V=800.0 PL=0
MOVL C00266 V=800.0 PL=0
MOVL C00267 V=800.0 PL=0
MOVL C00268 V=800.0 PL=0
MOVL C00269 V=800.0 PL=0
MOVL C00270 V=800.0 PL=0
MOVL C00271 V=800.0 PL=0
MOVL C00272 V=800.0 PL=0
MOVL C00273 V=800.0 PL=0
MOVL C00274 V=800.0 PL=0
MOVL C00275 V=800.0 PL=0
MOVL C00276 V=800.0 PL=0
MOVL C00277 V=800.0 PL=0
MOVL C00278 V=800.0 PL=0
MOVL C00279 V=800.0 PL=0
MOVL C00280 V=800.0 PL=0
MOVL C00281 V=800.0 PL=0
MOVL C00282 V=800.0 PL=0
MOVL C00283 V=800.0 PL=0
MOVL C00284 V=800.0 PL=0
MOVL C00285 V=800.0 PL=0
MOVL C00286 V=800.0 PL=0
MOVL C00287 V=800.0 PL=0
MOVL C00288 V=800.0 PL=0
MOVL C00289 V=800.0 PL=0
MOVL C00290 V=800.0 PL=0
MOVL C00291 V=800.0 PL=0
MOVL C00292 V=800.0 PL=0
MOVL C00293 V=800.0 PL=0
MOVL C00294 V=800.0 PL=0
MOVL C00295 V=800.0 PL=0
MOVL C00296 V=800.0 PL=0
MOVL C00297 V=800.0 PL=0
MOVL C00298 V=800.0 PL=0
MOVL C00299 V=800.0 PL=0
MOVL C00300 V=800.0 PL=0
MOVL C00301 V=800.0 PL=0
MOVL C00302 V=800.0 PL=0
MOVL C00303 V=800.0 PL=0
MOVL C00304 V=800.0 PL=0
MOVL C00305 V=800.0 PL=0
MOVL C00306 V=800.0 PL=0
MOVL C00307 V=800.0 PL=0
MOVL C00308 V=800.0 PL=0
MOVL C00309 V=800.0 PL=0
MOVL C00310 V=800.0 PL=0
MOVL C00311 V=800.0 PL=0
MOVL C00312 V=800.0 PL=0
MOVL C00313 V=800.0 PL=0
MOVL C00314 V=800.0 PL=0
MOVL C00315 V=800.0 PL=0
MOVL C00316 V=800.0 PL=0
MOVL C00317 V=800.0 PL=0
MOVL C00318 V=800.0 PL=0
MOVL C00319 V=800.0 PL=0
MOVL C00320 V=800.0 PL=0
MOVL C00321 V=800.0 PL=0
MOVL C00322 V=800.0 PL=0
MOVL C00323 V=800.0 PL=0
MOVL C00324 V=800.0 PL=0
MOVL C00325 V=800.0 PL=0
MOVL C00326 V=800.0 PL=0
MOVL C00327 V=800.0 PL=0
MOVL C00328 V=800.0 PL=0
MOVL C00329 V=800.0 PL=0
MOVL C00330 V=800.0 PL=0
MOVL C00331 V=800.0 PL=0
MOVL C00332 V=800.0 PL=0
MOVL C00333 V=800.0 PL=0
MOVL C00334 V=800.0 PL=0
MOVL C00335 V=800.0 PL=0
MOVL C00336 V=800.0 PL=0
MOVL C00337 V=800.0 PL=0
MOVL C00338 V=800.0 PL=0
MOVL C00339 V=800.0 PL=0
MOVL C00340 V=800.0 PL=0
MOVL C00341 V=800.0 PL=0
MOVL C00342 V=800.0 PL=0
MOVL C00343 V=800.0 PL=0
MOVL C00344 V=800.0 PL=0
MOVL C00345 V=800.0 PL=0
MOVL C00346 V=800.0 PL=0
MOVL C00347 V=800.0 PL=0
MOVL C00348 V=800.0 PL=0
MOVL C00349 V=800.0 PL=0
MOVL C00350 V=800.0 PL=0
MOVL C00351 V=800.0 PL=0
MOVL C00352 V=800.0 PL=0
MOVL C00353 V=800.0 PL=0
MOVL C00354 V=800.0 PL=0
MOVL C00355 V=800.0 PL=0
MOVL C00356 V=800.0 PL=0
MOVL C00357 V=800.0 PL=0
MOVL C00358 V=800.0 PL=0
MOVL C00359 V=800.0 PL=0
MOVL C00360 V=800.0 PL=0
MOVL C00361 V=800.0 PL=0
MOVL C00362 V=800.0 PL=0
MOVL C00363 V=800.0 PL=0
MOVL C00364 V=800.0 PL=0
MOVL C00365 V=800.0 PL=0
MOVL C00366 V=800.0 PL=0
MOVL C00367 V=800.0 PL=0
MOVL C00368 V=800.0 PL=0
MOVL C00369 V=800.0 PL=0
MOVL C00370 V=800.0 PL=0
MOVL C00371 V=800.0 PL=0
MOVL C00372 V=800.0 PL=0
MOVL C00373 V=800.0 PL=0
MOVL C00374 V=800.0 PL=0
MOVL C00375 V=800.0 PL=0
MOVL C00376 V=800.0 PL=0
MOVL C00377 V=800.0 PL=0
MOVL C00378 V=800.0 PL=0
MOVL C00379 V=800.0 PL=0
MOVL C00380 V=800.0 PL=0
MOVL C00381 V=800.0 PL=0
MOVL C00382 V=800.0 PL=0
MOVL C00383 V=800.0 PL=0
MOVL C00384 V=800.0 PL=0
MOVL C00385 V=800.0 PL=0
MOVL C00386 V=800.0 PL=0
MOVL C00387 V=800.0 PL=0
MOVL C00388 V=800.0 PL=0
MOVL C00389 V=800.0 PL=0
MOVL C00390 V=800.0 PL=0
MOVL C00391 V=800.0 PL=0
MOVL C00392 V=800.0 PL=0
MOVL C00393 V=800.0 PL=0
MOVL C00394 V=800.0 PL=0
MOVL C00395 V=800.0 PL=0
MOVL C00396 V=800.0 PL=0
MOVL C00397 V=800.0 PL=0
MOVL C00398 V=800.0 PL=0
MOVL C00399 V=800.0 PL=0
MOVL C00400 V=800.0 PL=0
MOVL C00401 V=800.0 PL=0
MOVL C00402 V=800.0 PL=0
MOVL C00403 V=800.0 PL=0
MOVL C00404 V=800.0 PL=0
MOVL C00405 V=800.0 PL=0
MOVL C00406 V=800.0 PL=0
MOVL C00407 V=800.0 PL=0
MOVL C00408 V=800.0 PL=0
MOVL C00409 V=800.0 PL=0
MOVL C00410 V=800.0 PL=0
MOVL C00411 V=800.0 PL=0
MOVL C00412 V=800.0 PL=0
MOVL C00413 V=800.0 PL=0
MOVL C00414 V=800.0 PL=0
MOVL C00415 V=800.0 PL=0
MOVL C00416 V=800.0 PL=0
MOVL C00417 V=800.0 PL=0
MOVL C00418 V=800.0 PL=0
MOVL C00419 V=800.0 PL=0
MOVL C00420 V=800.0 PL=0
MOVL C00421 V=800.0 PL=0
MOVL C00422 V=800.0 PL=0
MOVL C00423 V=800.0 PL=0
MOVL C00424 V=800.0 PL=0
MOVL C00425 V=800.0 PL=0
MOVL C00426 V=800.0 PL=0
MOVL C00427 V=800.0 PL=0
MOVL C00428 V=800.0 PL=0
MOVL C00429 V=800.0 PL=0
MOVL C00430 V=800.0 PL=0
MOVL C00431 V=800.0 PL=0
MOVL C00432 V=800.0 PL=0
MOVL C00433 V=800.0 PL=0
MOVL C00434 V=800.0 PL=0
MOVL C00435 V=800.0 PL=0
MOVL C00436 V=800.0 PL=0
MOVL C00437 V=800.0 PL=0
MOVL C00438 V=800.0 PL=0
MOVL C00439 V=800.0 PL=0
MOVL C00440 V=800.0 PL=0
MOVL C00441 V=800.0 PL=0
MOVL C00442 V=800.0 PL=0
MOVL C00443 V=800.0 PL=0
MOVL C00444 V=800.0 PL=0
MOVL C00445 V=800.0 PL=0
MOVL C00446 V=800.0 PL=0
MOVL C00447 V=800.0 PL=0
MOVL C00448 V=800.0 PL=0
MOVL C00449 V=800.0 PL=0
MOVL C00450 V=800.0 PL=0
MOVL C00451 V=800.0 PL=0
MOVL C00452 V=800.0 PL=0
MOVL C00453 V=800.0 PL=0
MOVL C00454 V=800.0 PL=0
MOVL C00455 V=800.0 PL=0
MOVL C00456 V=800.0 PL=0
MOVL C00457 V=800.0 PL=0
MOVL C00458 V=800.0 PL=0
MOVL C00459 V=800.0 PL=0
MOVL C00460 V=800.0 PL=0
MOVL C00461 V=800.0 PL=0
MOVL C00462 V=800.0 PL=0
MOVL C00463 V=800.0 PL=0
MOVL C00464 V=800.0 PL=0
MOVL C00465 V=800.0 PL=0
MOVL C00466 V=800.0 PL=0
MOVL C00467 V=800.0 PL=0
MOVL C00468 V=800.0 PL=0
MOVL C00469 V=800.0 PL=0
MOVL C00470 V=800.0 PL=0
MOVL C00471 V=800.0 PL=0
MOVL C00472 V=800.0 PL=0
MOVL C00473 V=800.0 PL=0
MOVL C00474 V=800.0 PL=0
MOVL C00475 V=800.0 PL=0
MOVL C00476 V=800.0 PL=0
MOVL C00477 V=800.0 PL=0
MOVL C00478 V=800.0 PL=0
MOVL C00479 V=800.0 PL=0
MOVL C00480 V=800.0 PL=0
MOVL C00481 V=800.0 PL=0
MOVL C00482 V=800.0 PL=0
MOVL C00483 V=800.0 PL=0
MOVL C00484 V=800.0 PL=0
MOVL C00485 V=800.0 PL=0
MOVL C00486 V=800.0 PL=0
MOVL C00487 V=800.0 PL=0
MOVL C00488 V=800.0 PL=0
MOVL C00489 V=800.0 PL=0
MOVL C00490 V=800.0 PL=0
MOVL C00491 V=800.0 PL=0
MOVL C00492 V=800.0 PL=0
MOVL C00493 V=800.0 PL=0
MOVL C00494 V=800.0 PL=0
MOVL C00495 V=800.0 PL=0
MOVL C00496 V=800.0 PL=0
MOVL C00497 V=800.0 PL=0
MOVL C00498 V=800.0 PL=0
MOVL C00499 V=800.0 PL=0
MOVL C00500 V=800.0 PL=0
MOVL C00501 V=800.0 PL=0
MOVL C00502 V=800.0 PL=0
MOVL C00503 V=800.0 PL=0
MOVL C00504 V=800.0 PL=0
MOVL C00505 V=800.0 PL=0
MOVL C00506 V=800.0 PL=0
MOVL C00507 V=800.0 PL=0
MOVL C00508 V=800.0 PL=0
MOVL C00509 V=800.0 PL=0
MOVL C00510 V=800.0 PL=0
MOVL C00511 V=800.0 PL=0
MOVL C00512 V=800.0 PL=0
MOVL C00513 V=800.0 PL=0
MOVL C00514 V=800.0 PL=0
MOVL C00515 V=800.0 PL=0
MOVL C00516 V=800.0 PL=0
MOVL C00517 V=800.0 PL=0
MOVL C00518 V=800.0 PL=0
MOVL C00519 V=800.0 PL=0
MOVL C00520 V=800.0 PL=0
MOVL C00521 V=800.0 PL=0
MOVL C00522 V=800.0 PL=0
MOVL C00523 V=800.0 PL=0
MOVL C00524 V=800.0 PL=0
MOVL C00525 V=800.0 PL=0
MOVL C00526 V=800.0 PL=0
MOVL C00527 V=800.0 PL=0
MOVL C00528 V=800.0 PL=0
MOVL C00529 V=800.0 PL=0
MOVL C00530 V=800.0 PL=0
MOVL C00531 V=800.0 PL=0
MOVL C00532 V=800.0 PL=0
MOVL C00533 V=800.0 PL=0
MOVL C00534 V=800.0 PL=0
MOVL C00535 V=800.0 PL=0
MOVL C00536 V=800.0 PL=0
MOVL C00537 V=800.0 PL=0
MOVL C00538 V=800.0 PL=0
MOVL C00539 V=800.0 PL=0
MOVL C00540 V=800.0 PL=0
MOVL C00541 V=800.0 PL=0
MOVL C00542 V=800.0 PL=0
MOVL C00543 V=800.0 PL=0
MOVL C00544 V=800.0 PL=0
MOVL C00545 V=800.0 PL=0
MOVL C00546 V=800.0 PL=0
MOVL C00547 V=800.0 PL=0
MOVL C00548 V=800.0 PL=0
MOVL C00549 V=800.0 PL=0
MOVL C00550 V=800.0 PL=0
MOVL C00551 V=800.0 PL=0
MOVL C00552 V=800.0 PL=0
MOVL C00553 V=800.0 PL=0
MOVL C00554 V=800.0 PL=0
MOVL C00555 V=800.0 PL=0
MOVL C00556 V=800.0 PL=0
MOVL C00557 V=800.0 PL=0
MOVL C00558 V=800.0 PL=0
MOVL C00559 V=800.0 PL=0
MOVL C00560 V=800.0 PL=0
MOVL C00561 V=800.0 PL=0
MOVL C00562 V=800.0 PL=0
MOVL C00563 V=800.0 PL=0
MOVL C00564 V=800.0 PL=0
MOVL C00565 V=800.0 PL=0
MOVL C00566 V=800.0 PL=0
MOVL C00567 V=800.0 PL=0
MOVL C00568 V=800.0 PL=0
MOVL C00569 V=800.0 PL=0
MOVL C00570 V=800.0 PL=0
MOVL C00571 V=800.0 PL=0
MOVL C00572 V=800.0 PL=0
MOVL C00573 V=800.0 PL=0
MOVL C00574 V=800.0 PL=0
MOVL C00575 V=800.0 PL=0
MOVL C00576 V=800.0 PL=0
MOVL C00577 V=800.0 PL=0
MOVL C00578 V=800.0 PL=0
MOVL C00579 V=800.0 PL=0
MOVL C00580 V=800.0 PL=0
MOVL C00581 V=800.0 PL=0
MOVL C00582 V=800.0 PL=0
MOVL C00583 V=800.0 PL=0
MOVL C00584 V=800.0 PL=0
MOVL C00585 V=800.0 PL=0
MOVL C00586 V=800.0 PL=0
MOVL C00587 V=800.0 PL=0
MOVL C00588 V=800.0 PL=0
MOVL C00589 V=800.0 PL=0
MOVL C00590 V=800.0 PL=0
MOVL C00591 V=800.0 PL=0
MOVL C00592 V=800.0 PL=0
MOVL C00593 V=800.0 PL=0
MOVL C00594 V=800.0 PL=0
MOVL C00595 V=800.0 PL=0
MOVL C00596 V=800.0 PL=0
MOVL C00597 V=800.0 PL=0
MOVL C00598 V=800.0 PL=0
MOVL C00599 V=800.0 PL=0
MOVL C00600 V=800.0 PL=0
MOVL C00601 V=800.0 PL=0
MOVL C00602 V=800.0 PL=0
MOVL C00603 V=800.0 PL=0
MOVL C00604 V=800.0 PL=0
MOVL C00605 V=800.0 PL=0
MOVL C00606 V=800.0 PL=0
MOVL C00607 V=800.0 PL=0
MOVL C00608 V=800.0 PL=0
MOVL C00609 V=800.0 PL=0
MOVL C00610 V=800.0 PL=0
MOVL C00611 V=800.0 PL=0
MOVL C00612 V=800.0 PL=0
MOVL C00613 V=800.0 PL=0
MOVL C00614 V=800.0 PL=0
MOVL C00615 V=800.0 PL=0
MOVL C00616 V=800.0 PL=0
MOVL C00617 V=800.0 PL=0
MOVL C00618 V=800.0 PL=0
MOVL C00619 V=800.0 PL=0
MOVL C00620 V=800.0 PL=0
MOVL C00621 V=800.0 PL=0
MOVL C00622 V=800.0 PL=0
MOVL C00623 V=800.0 PL=0
MOVL C00624 V=800.0 PL=0
MOVL C00625 V=800.0 PL=0
MOVL C00626 V=800.0 PL=0
MOVL C00627 V=800.0 PL=0
MOVL C00628 V=800.0 PL=0
MOVL C00629 V=800.0 PL=0
MOVL C00630 V=800.0 PL=0
MOVL C00631 V=800.0 PL=0
MOVL C00632 V=800.0 PL=0
MOVL C00633 V=800.0 PL=0
MOVL C00634 V=800.0 PL=0
MOVL C00635 V=800.0 PL=0
MOVL C00636 V=800.0 PL=0
MOVL C00637 V=800.0 PL=0
MOVL C00638 V=800.0 PL=0
MOVL C00639 V=800.0 PL=0
MOVL C00640 V=800.0 PL=0
MOVL C00641 V=800.0 PL=0
MOVL C00642 V=800.0 PL=0
MOVL C00643 V=800.0 PL=0
MOVL C00644 V=800.0 PL=0
MOVL C00645 V=800.0 PL=0
MOVL C00646 V=800.0 PL=0
MOVL C00647 V=800.0 PL=0
MOVL C00648 V=800.0 PL=0
MOVL C00649 V=800.0 PL=0
MOVL C00650 V=800.0 PL=0
MOVL C00651 V=800.0 PL=0
MOVL C00652 V=800.0 PL=0
MOVL C00653 V=800.0 PL=0
MOVL C00654 V=800.0 PL=0
MOVL C00655 V=800.0 PL=0
MOVL C00656 V=800.0 PL=0
MOVL C00657 V=800.0 PL=0
MOVL C00658 V=800.0 PL=0
MOVL C00659 V=800.0 PL=0
MOVL C00660 V=800.0 PL=0
MOVL C00661 V=800.0 PL=0
MOVL C00662 V=800.0 PL=0
MOVL C00663 V=800.0 PL=0
MOVL C00664 V=800.0 PL=0
MOVL C00665 V=800.0 PL=0
MOVL C00666 V=800.0 PL=0
MOVL C00667 V=800.0 PL=0
MOVL C00668 V=800.0 PL=0
MOVL C00669 V=800.0 PL=0
MOVL C00670 V=800.0 PL=0
MOVL C00671 V=800.0 PL=0
MOVL C00672 V=800.0 PL=0
MOVL C00673 V=800.0 PL=0
MOVL C00674 V=800.0 PL=0
MOVL C00675 V=800.0 PL=0
MOVL C00676 V=800.0 PL=0
MOVL C00677 V=800.0 PL=0
MOVL C00678 V=800.0 PL=0
MOVL C00679 V=800.0 PL=0
MOVL C00680 V=800.0 PL=0
MOVL C00681 V=800.0 PL=0
MOVL C00682 V=800.0 PL=0
MOVL C00683 V=800.0 PL=0
MOVL C00684 V=800.0 PL=0
MOVL C00685 V=800.0 PL=0
MOVL C00686 V=800.0 PL=0
MOVL C00687 V=800.0 PL=0
MOVL C00688 V=800.0 PL=0
MOVL C00689 V=800.0 PL=0
MOVL C00690 V=800.0 PL=0
MOVL C00691 V=800.0 PL=0
MOVL C00692 V=800.0 PL=0
MOVL C00693 V=800.0 PL=0
MOVL C00694 V=800.0 PL=0
MOVL C00695 V=800.0 PL=0
MOVL C00696 V=800.0 PL=0
MOVL C00697 V=800.0 PL=0
MOVL C00698 V=800.0 PL=0
MOVL C00699 V=800.0 PL=0
MOVL C00700 V=800.0 PL=0
MOVL C00701 V=800.0 PL=0
MOVL C00702 V=800.0 PL=0
MOVL C00703 V=800.0 PL=0
MOVL C00704 V=800.0 PL=0
MOVL C00705 V=800.0 PL=0
MOVL C00706 V=800.0 PL=0
MOVL C00707 V=800.0 PL=0
MOVL C00708 V=800.0 PL=0
MOVL C00709 V=800.0 PL=0
MOVL C00710 V=800.0 PL=0
MOVL C00711 V=800.0 PL=0
MOVL C00712 V=800.0 PL=0
MOVL C00713 V=800.0 PL=0
MOVL C00714 V=800.0 PL=0
MOVL C00715 V=800.0 PL=0
MOVL C00716 V=800.0 PL=0
MOVL C00717 V=800.0 PL=0
MOVL C00718 V=800.0 PL=0
MOVL C00719 V=800.0 PL=0
MOVL C00720 V=800.0 PL=0
MOVL C00721 V=800.0 PL=0
MOVL C00722 V=800.0 PL=0
MOVL C00723 V=800.0 PL=0
MOVL C00724 V=800.0 PL=0
MOVL C00725 V=800.0 PL=0
MOVL C00726 V=800.0 PL=0
MOVL C00727 V=800.0 PL=0
MOVL C00728 V=800.0 PL=0
MOVL C00729 V=800.0 PL=0
MOVL C00730 V=800.0 PL=0
MOVL C00731 V=800.0 PL=0
MOVL C00732 V=800.0 PL=0
MOVL C00733 V=800.0 PL=0
MOVL C00734 V=800.0 PL=0
MOVL C00735 V=800.0 PL=0
MOVL C00736 V=800.0 PL=0
MOVL C00737 V=800.0 PL=0
MOVL C00738 V=800.0 PL=0
MOVL C00739 V=800.0 PL=0
MOVL C00740 V=800.0 PL=0
MOVL C00741 V=800.0 PL=0
MOVL C00742 V=800.0 PL=0
MOVL C00743 V=800.0 PL=0
MOVL C00744 V=800.0 PL=0
MOVL C00745 V=800.0 PL=0
MOVL C00746 V=800.0 PL=0
MOVL C00747 V=800.0 PL=0
MOVL C00748 V=800.0 PL=0
MOVL C00749 V=800.0 PL=0
MOVL C00750 V=800.0 PL=0
MOVL C00751 V=800.0 PL=0
MOVL C00752 V=800.0 PL=0
MOVL C00753 V=800.0 PL=0
MOVL C00754 V=800.0 PL=0
MOVL C00755 V=800.0 PL=0
MOVL C00756 V=800.0 PL=0
MOVL C00757 V=800.0 PL=0
MOVL C00758 V=800.0 PL=0
MOVL C00759 V=800.0 PL=0
MOVL C00760 V=800.0 PL=0
MOVL C00761 V=800.0 PL=0
MOVL C00762 V=800.0 PL=0
MOVL C00763 V=800.0 PL=0
MOVL C00764 V=800.0 PL=0
MOVL C00765 V=800.0 PL=0
MOVL C00766 V=800.0 PL=0
MOVL C00767 V=800.0 PL=0
MOVL C00768 V=800.0 PL=0
MOVL C00769 V=800.0 PL=0
MOVL C00770 V=800.0 PL=0
MOVL C00771 V=800.0 PL=0
MOVL C00772 V=800.0 PL=0
MOVL C00773 V=800.0 PL=0
MOVL C00774 V=800.0 PL=0
MOVL C00775 V=800.0 PL=0
MOVL C00776 V=800.0 PL=0
MOVL C00777 V=800.0 PL=0
MOVL C00778 V=800.0 PL=0
MOVL C00779 V=800.0 PL=0
MOVL C00780 V=800.0 PL=0
MOVL C00781 V=800.0 PL=0
MOVL C00782 V=800.0 PL=0
MOVL C00783 V=800.0 PL=0
MOVL C00784 V=800.0 PL=0
MOVL C00785 V=800.0 PL=0
MOVL C00786 V=800.0 PL=0
MOVL C00787 V=800.0 PL=0
MOVL C00788 V=800.0 PL=0
MOVL C00789 V=800.0 PL=0
MOVL C00790 V=800.0 PL=0
MOVL C00791 V=800.0 PL=0
MOVL C00792 V=800.0 PL=0
MOVL C00793 V=800.0 PL=0
MOVL C00794 V=800.0 PL=0
MOVL C00795 V=800.0 PL=0
MOVL C00796 V=800.0 PL=0
MOVL C00797 V=800.0 PL=0
MOVL C00798 V=800.0 PL=0
MOVL C00799 V=800.0 PL=0
MOVL C00800 V=800.0 PL=0
MOVL C00801 V=800.0 PL=0
MOVL C00802 V=800.0 PL=0
MOVL C00803 V=800.0 PL=0
MOVL C00804 V=800.0 PL=0
MOVL C00805 V=800.0 PL=0
MOVL C00806 V=800.0 PL=0
MOVL C00807 V=800.0 PL=0
MOVL C00808 V=800.0 PL=0
MOVL C00809 V=800.0 PL=0
MOVL C00810 V=800.0 PL=0
MOVL C00811 V=800.0 PL=0
MOVL C00812 V=800.0 PL=0
MOVL C00813 V=800.0 PL=0
MOVL C00814 V=800.0 PL=0
MOVL C00815 V=800.0 PL=0
MOVL C00816 V=800.0 PL=0
MOVL C00817 V=800.0 PL=0
MOVL C00818 V=800.0 PL=0
MOVL C00819 V=800.0 PL=0
MOVL C00820 V=800.0 PL=0
MOVL C00821 V=800.0 PL=0
MOVL C00822 V=800.0 PL=0
MOVL C00823 V=800.0 PL=0
MOVL C00824 V=800.0 PL=0
MOVL C00825 V=800.0 PL=0
MOVL C00826 V=800.0 PL=0
MOVL C00827 V=800.0 PL=0
MOVL C00828 V=800.0 PL=0
MOVL C00829 V=800.0 PL=0
MOVL C00830 V=800.0 PL=0
MOVL C00831 V=800.0 PL=0
MOVL C00832 V=800.0 PL=0
MOVL C00833 V=800.0 PL=0
MOVL C00834 V=800.0 PL=0
MOVL C00835 V=800.0 PL=0
MOVL C00836 V=800.0 PL=0
MOVL C00837 V=800.0 PL=0
MOVL C00838 V=800.0 PL=0
MOVL C00839 V=800.0 PL=0
MOVL C00840 V=800.0 PL=0
MOVL C00841 V=800.0 PL=0
MOVL C00842 V=800.0 PL=0
MOVL C00843 V=800.0 PL=0
MOVL C00844 V=800.0 PL=0
MOVL C00845 V=800.0 PL=0
MOVL C00846 V=800.0 PL=0
MOVL C00847 V=800.0 PL=0
MOVL C00848 V=800.0 PL=0
MOVL C00849 V=800.0 PL=0
MOVL C00850 V=800.0 PL=0
MOVL C00851 V=800.0 PL=0
MOVL C00852 V=800.0 PL=0
MOVL C00853 V=800.0 PL=0
MOVL C00854 V=800.0 PL=0
MOVL C00855 V=800.0 PL=0
MOVL C00856 V=800.0 PL=0
MOVL C00857 V=800.0 PL=0
MOVL C00858 V=800.0 PL=0
MOVL C00859 V=800.0 PL=0
MOVL C00860 V=800.0 PL=0
MOVL C00861 V=800.0 PL=0
MOVL C00862 V=800.0 PL=0
MOVL C00863 V=800.0 PL=0
MOVL C00864 V=800.0 PL=0
MOVL C00865 V=800.0 PL=0
MOVL C00866 V=800.0 PL=0
MOVL C00867 V=800.0 PL=0
MOVL C00868 V=800.0 PL=0
MOVL C00869 V=800.0 PL=0
MOVL C00870 V=800.0 PL=0
MOVL C00871 V=800.0 PL=0
MOVL C00872 V=800.0 PL=0
MOVL C00873 V=800.0 PL=0
MOVL C00874 V=800.0 PL=0
MOVL C00875 V=800.0 PL=0
MOVL C00876 V=800.0 PL=0
MOVL C00877 V=800.0 PL=0
MOVL C00878 V=800.0 PL=0
MOVL C00879 V=800.0 PL=0
MOVL C00880 V=800.0 PL=0
MOVL C00881 V=800.0 PL=0
MOVL C00882 V=800.0 PL=0
MOVL C00883 V=800.0 PL=0
MOVL C00884 V=800.0 PL=0
MOVL C00885 V=800.0 PL=0
MOVL C00886 V=800.0 PL=0
MOVL C00887 V=800.0 PL=0
MOVL C00888 V=800.0 PL=0
MOVL C00889 V=800.0 PL=0
MOVL C00890 V=800.0 PL=0
MOVL C00891 V=800.0 PL=0
MOVL C00892 V=800.0 PL=0
MOVL C00893 V=800.0 PL=0
MOVL C00894 V=800.0 PL=0
MOVL C00895 V=800.0 PL=0
MOVL C00896 V=800.0 PL=0
MOVL C00897 V=800.0 PL=0
MOVL C00898 V=800.0 PL=0
MOVL C00899 V=800.0 PL=0
MOVL C00900 V=800.0 PL=0
MOVL C00901 V=800.0 PL=0
MOVL C00902 V=800.0 PL=0
MOVL C00903 V=800.0 PL=0
MOVL C00904 V=800.0 PL=0
MOVL C00905 V=800.0 PL=0
MOVL C00906 V=800.0 PL=0
MOVL C00907 V=800.0 PL=0
MOVL C00908 V=800.0 PL=0
MOVL C00909 V=800.0 PL=0
MOVL C00910 V=800.0 PL=0
MOVL C00911 V=800.0 PL=0
MOVL C00912 V=800.0 PL=0
MOVL C00913 V=800.0 PL=0
MOVL C00914 V=800.0 PL=0
MOVL C00915 V=800.0 PL=0
MOVL C00916 V=800.0 PL=0
MOVL C00917 V=800.0 PL=0
MOVL C00918 V=800.0 PL=0
MOVL C00919 V=800.0 PL=0
MOVL C00920 V=800.0 PL=0
MOVL C00921 V=800.0 PL=0
MOVL C00922 V=800.0 PL=0
MOVL C00923 V=800.0 PL=0
MOVL C00924 V=800.0 PL=0
MOVL C00925 V=800.0 PL=0
MOVL C00926 V=800.0 PL=0
MOVL C00927 V=800.0 PL=0
MOVL C00928 V=800.0 PL=0
MOVL C00929 V=800.0 PL=0
MOVL C00930 V=800.0 PL=0
MOVL C00931 V=800.0 PL=0
MOVL C00932 V=800.0 PL=0
MOVL C00933 V=800.0 PL=0
MOVL C00934 V=800.0 PL=0
MOVL C00935 V=800.0 PL=0
MOVL C00936 V=800.0 PL=0
MOVL C00937 V=800.0 PL=0
MOVL C00938 V=800.0 PL=0
MOVL C00939 V=800.0 PL=0
MOVL C00940 V=800.0 PL=0
MOVL C00941 V=800.0 PL=0
MOVL C00942 V=800.0 PL=0
MOVL C00943 V=800.0 PL=0
MOVL C00944 V=800.0 PL=0
MOVL C00945 V=800.0 PL=0
MOVL C00946 V=800.0 PL=0
MOVL C00947 V=800.0 PL=0
MOVL C00948 V=800.0 PL=0
MOVL C00949 V=800.0 PL=0
MOVL C00950 V=800.0 PL=0
MOVL C00951 V=800.0 PL=0
MOVL C00952 V=800.0 PL=0
MOVL C00953 V=800.0 PL=0
MOVL C00954 V=800.0 PL=0
MOVL C00955 V=800.0 PL=0
MOVL C00956 V=800.0 PL=0
MOVL C00957 V=800.0 PL=0
MOVL C00958 V=800.0 PL=0
MOVL C00959 V=800.0 PL=0
MOVL C00960 V=800.0 PL=0
MOVL C00961 V=800.0 PL=0
MOVL C00962 V=800.0 PL=0
MOVL C00963 V=800.0 PL=0
MOVL C00964 V=800.0 PL=0
MOVL C00965 V=800.0 PL=0
MOVL C00966 V=800.0 PL=0
MOVL C00967 V=800.0 PL=0
MOVL C00968 V=800.0 PL=0
MOVL C00969 V=800.0 PL=0
MOVL C00970 V=800.0 PL=0
MOVL C00971 V=800.0 PL=0
MOVL C00972 V=800.0 PL=0
MOVL C00973 V=800.0 PL=0
MOVL C00974 V=800.0 PL=0
MOVL C00975 V=800.0 PL=0
MOVL C00976 V=800.0 PL=0
MOVL C00977 V=800.0 PL=0
MOVL C00978 V=800.0 PL=0
MOVL C00979 V=800.0 PL=0
MOVL C00980 V=800.0 PL=0
MOVL C00981 V=800.0 PL=0
MOVL C00982 V=800.0 PL=0
MOVL C00983 V=800.0 PL=0
MOVL C00984 V=800.0 PL=0
MOVL C00985 V=800.0 PL=0
MOVL C00986 V=800.0 PL=0
MOVL C00987 V=800.0 PL=0
MOVL C00988 V=800.0 PL=0
MOVL C00989 V=800.0 PL=0
MOVL C00990 V=800.0 PL=0
MOVL C00991 V=800.0 PL=0
MOVL C00992 V=800.0 PL=0
MOVL C00993 V=800.0 PL=0
MOVL C00994 V=800.0 PL=0
MOVL C00995 V=800.0 PL=0
MOVL C00996 V=800.0 PL=0
MOVL C00997 V=800.0 PL=0
MOVL C00998 V=800.0 PL=0
MOVL C00999 V=800.0 PL=0
MOVL C01000 V=800.0 PL=0
MOVL C01001 V=800.0 PL=0
MOVL C01002 V=800.0 PL=0
MOVL C01003 V=800.0 PL=0
MOVL C01004 V=800.0 PL=0
MOVL C01005 V=800.0 PL=0
MOVL C01006 V=800.0 PL=0
MOVL C01007 V=800.0 PL=0
MOVL C01008 V=800.0 PL=0
MOVL C01009 V=800.0 PL=0
MOVL C01010 V=800.0 PL=0
MOVL C01011 V=800.0 PL=0
MOVL C01012 V=800.0 PL=0
MOVL C01013 V=800.0 PL=0
MOVL C01014 V=800.0 PL=0
MOVL C01015 V=800.0 PL=0
MOVL C01016 V=800.0 PL=0
MOVL C01017 V=800.0 PL=0
MOVL C01018 V=800.0 PL=0
MOVL C01019 V=800.0 PL=0
MOVL C01020 V=800.0 PL=0
MOVL C01021 V=800.0 PL=0
MOVL C01022 V=800.0 PL=0
MOVL C01023 V=800.0 PL=0
MOVL C01024 V=800.0 PL=0
MOVL C01025 V=800.0 PL=0
MOVL C01026 V=800.0 PL=0
MOVL C01027 V=800.0 PL=0
MOVL C01028 V=800.0 PL=0
MOVL C01029 V=800.0 PL=0
MOVL C01030 V=800.0 PL=0
MOVL C01031 V=800.0 PL=0
MOVL C01032 V=800.0 PL=0
MOVL C01033 V=800.0 PL=0
MOVL C01034 V=800.0 PL=0
MOVL C01035 V=800.0 PL=0
MOVL C01036 V=800.0 PL=0
MOVL C01037 V=800.0 PL=0
MOVL C01038 V=800.0 PL=0
MOVL C01039 V=800.0 PL=0
MOVL C01040 V=800.0 PL=0
MOVL C01041 V=800.0 PL=0
MOVL C01042 V=800.0 PL=0
MOVL C01043 V=800.0 PL=0
MOVL C01044 V=800.0 PL=0
MOVL C01045 V=800.0 PL=0
MOVL C01046 V=800.0 PL=0
MOVL C01047 V=800.0 PL=0
MOVL C01048 V=800.0 PL=0
MOVL C01049 V=800.0 PL=0
MOVL C01050 V=800.0 PL=0
MOVL C01051 V=800.0 PL=0
MOVL C01052 V=800.0 PL=0
MOVL C01053 V=800.0 PL=0
MOVL C01054 V=800.0 PL=0
MOVL C01055 V=800.0 PL=0
MOVL C01056 V=800.0 PL=0
MOVL C01057 V=800.0 PL=0
MOVL C01058 V=800.0 PL=0
MOVL C01059 V=800.0 PL=0
MOVL C01060 V=800.0 PL=0
MOVL C01061 V=800.0 PL=0
MOVL C01062 V=800.0 PL=0
MOVL C01063 V=800.0 PL=0
MOVL C01064 V=800.0 PL=0
MOVL C01065 V=800.0 PL=0
MOVL C01066 V=800.0 PL=0
MOVL C01067 V=800.0 PL=0
MOVL C01068 V=800.0 PL=0
MOVL C01069 V=800.0 PL=0
MOVL C01070 V=800.0 PL=0
MOVL C01071 V=800.0 PL=0
MOVL C01072 V=800.0 PL=0
MOVL C01073 V=800.0 PL=0
MOVL C01074 V=800.0 PL=0
MOVL C01075 V=800.0 PL=0
MOVL C01076 V=800.0 PL=0
MOVL C01077 V=800.0 PL=0
MOVL C01078 V=800.0 PL=0
MOVL C01079 V=800.0 PL=0
MOVL C01080 V=800.0 PL=0
MOVL C01081 V=800.0 PL=0
MOVL C01082 V=800.0 PL=0
MOVL C01083 V=800.0 PL=0
MOVL C01084 V=800.0 PL=0
MOVL C01085 V=800.0 PL=0
MOVL C01086 V=800.0 PL=0
MOVL C01087 V=800.0 PL=0
MOVL C01088 V=800.0 PL=0
MOVL C01089 V=800.0 PL=0
MOVL C01090 V=800.0 PL=0
MOVL C01091 V=800.0 PL=0
MOVL C01092 V=800.0 PL=0
MOVL C01093 V=800.0 PL=0
MOVL C01094 V=800.0 PL=0
MOVL C01095 V=800.0 PL=0
MOVL C01096 V=800.0 PL=0
MOVL C01097 V=800.0 PL=0
MOVL C01098 V=800.0 PL=0
MOVL C01099 V=800.0 PL=0
MOVL C01100 V=800.0 PL=0
MOVL C01101 V=800.0 PL=0
MOVL C01102 V=800.0 PL=0
MOVL C01103 V=800.0 PL=0
MOVL C01104 V=800.0 PL=0
MOVL C01105 V=800.0 PL=0
MOVL C01106 V=800.0 PL=0
MOVL C01107 V=800.0 PL=0
MOVL C01108 V=800.0 PL=0
MOVL C01109 V=800.0 PL=0
MOVL C01110 V=800.0 PL=0
MOVL C01111 V=800.0 PL=0
MOVL C01112 V=800.0 PL=0
MOVL C01113 V=800.0 PL=0
MOVL C01114 V=800.0 PL=0
MOVL C01115 V=800.0 PL=0
MOVL C01116 V=800.0 PL=0
MOVL C01117 V=800.0 PL=0
MOVL C01118 V=800.0 PL=0
MOVL C01119 V=800.0 PL=0
MOVL C01120 V=800.0 PL=0
MOVL C01121 V=800.0 PL=0
MOVL C01122 V=800.0 PL=0
MOVL C01123 V=800.0 PL=0
MOVL C01124 V=800.0 PL=0
MOVL C01125 V=800.0 PL=0
MOVL C01126 V=800.0 PL=0
MOVL C01127 V=800.0 PL=0
MOVL C01128 V=800.0 PL=0
MOVL C01129 V=800.0 PL=0
MOVL C01130 V=800.0 PL=0
MOVL C01131 V=800.0 PL=0
MOVL C01132 V=800.0 PL=0
MOVL C01133 V=800.0 PL=0
MOVL C01134 V=800.0 PL=0
MOVL C01135 V=800.0 PL=0
MOVL C01136 V=800.0 PL=0
MOVL C01137 V=800.0 PL=0
MOVL C01138 V=800.0 PL=0
MOVL C01139 V=800.0 PL=0
MOVL C01140 V=800.0 PL=0
MOVL C01141 V=800.0 PL=0
MOVL C01142 V=800.0 PL=0
MOVL C01143 V=800.0 PL=0
MOVL C01144 V=800.0 PL=0
MOVL C01145 V=800.0 PL=0
MOVL C01146 V=800.0 PL=0
MOVL C01147 V=800.0 PL=0
MOVL C01148 V=800.0 PL=0
MOVL C01149 V=800.0 PL=0
MOVL C01150 V=800.0 PL=0
MOVL C01151 V=800.0 PL=0
MOVL C01152 V=800.0 PL=0
MOVL C01153 V=800.0 PL=0
MOVL C01154 V=800.0 PL=0
MOVL C01155 V=800.0 PL=0
MOVL C01156 V=800.0 PL=0
MOVL C01157 V=800.0 PL=0
MOVL C01158 V=800.0 PL=0
MOVL C01159 V=800.0 PL=0
MOVL C01160 V=800.0 PL=0
MOVL C01161 V=800.0 PL=0
MOVL C01162 V=800.0 PL=0
MOVL C01163 V=800.0 PL=0
MOVL C01164 V=800.0 PL=0
MOVL C01165 V=800.0 PL=0
MOVL C01166 V=800.0 PL=0
MOVL C01167 V=800.0 PL=0
MOVL C01168 V=800.0 PL=0
MOVL C01169 V=800.0 PL=0
MOVL C01170 V=800.0 PL=0
MOVL C01171 V=800.0 PL=0
MOVL C01172 V=800.0 PL=0
MOVL C01173 V=800.0 PL=0
MOVL C01174 V=800.0 PL=0
MOVL C01175 V=800.0 PL=0
MOVL C01176 V=800.0 PL=0
MOVL C01177 V=800.0 PL=0
MOVL C01178 V=800.0 PL=0
MOVL C01179 V=800.0 PL=0
MOVL C01180 V=800.0 PL=0
MOVL C01181 V=800.0 PL=0
MOVL C01182 V=800.0 PL=0
MOVL C01183 V=800.0 PL=0
MOVL C01184 V=800.0 PL=0
MOVL C01185 V=800.0 PL=0
MOVL C01186 V=800.0 PL=0
MOVL C01187 V=800.0 PL=0
MOVL C01188 V=800.0 PL=0
MOVL C01189 V=800.0 PL=0
MOVL C01190 V=800.0 PL=0
MOVL C01191 V=800.0 PL=0
MOVL C01192 V=800.0 PL=0
MOVL C01193 V=800.0 PL=0
MOVL C01194 V=800.0 PL=0
MOVL C01195 V=800.0 PL=0
MOVL C01196 V=800.0 PL=0
MOVL C01197 V=800.0 PL=0
MOVL C01198 V=800.0 PL=0
MOVL C01199 V=800.0 PL=0
MOVL C01200 V=800.0 PL=0
MOVL C01201 V=800.0 PL=0
MOVL C01202 V=800.0 PL=0
MOVL C01203 V=800.0 PL=0
MOVL C01204 V=800.0 PL=0
MOVL C01205 V=800.0 PL=0
MOVL C01206 V=800.0 PL=0
MOVL C01207 V=800.0 PL=0
MOVL C01208 V=800.0 PL=0
MOVL C01209 V=800.0 PL=0
MOVL C01210 V=800.0 PL=0
MOVL C01211 V=800.0 PL=0
MOVL C01212 V=800.0 PL=0
MOVL C01213 V=800.0 PL=0
MOVL C01214 V=800.0 PL=0
MOVL C01215 V=800.0 PL=0
MOVL C01216 V=800.0 PL=0
MOVL C01217 V=800.0 PL=0
MOVL C01218 V=800.0 PL=0
MOVL C01219 V=800.0 PL=0
MOVL C01220 V=800.0 PL=0
MOVL C01221 V=800.0 PL=0
MOVL C01222 V=800.0 PL=0
MOVL C01223 V=800.0 PL=0
MOVL C01224 V=800.0 PL=0
MOVL C01225 V=800.0 PL=0
MOVL C01226 V=800.0 PL=0
MOVL C01227 V=800.0 PL=0
MOVL C01228 V=800.0 PL=0
MOVL C01229 V=800.0 PL=0
MOVL C01230 V=800.0 PL=0
MOVL C01231 V=800.0 PL=0
MOVL C01232 V=800.0 PL=0
MOVL C01233 V=800.0 PL=0
MOVL C01234 V=800.0 PL=0
MOVL C01235 V=800.0 PL=0
MOVL C01236 V=800.0 PL=0
MOVL C01237 V=800.0 PL=0
MOVL C01238 V=800.0 PL=0
MOVL C01239 V=800.0 PL=0
MOVL C01240 V=800.0 PL=0
MOVL C01241 V=800.0 PL=0
MOVL C01242 V=800.0 PL=0
MOVL C01243 V=800.0 PL=0
MOVL C01244 V=800.0 PL=0
MOVL C01245 V=800.0 PL=0
MOVL C01246 V=800.0 PL=0
MOVL C01247 V=800.0 PL=0
MOVL C01248 V=800.0 PL=0
MOVL C01249 V=800.0 PL=0
MOVL C01250 V=800.0 PL=0
MOVL C01251 V=800.0 PL=0
MOVL C01252 V=800.0 PL=0
MOVL C01253 V=800.0 PL=0
MOVL C01254 V=800.0 PL=0
MOVL C01255 V=800.0 PL=0
MOVL C01256 V=800.0 PL=0
MOVL C01257 V=800.0 PL=0
MOVL C01258 V=800.0 PL=0
MOVL C01259 V=800.0 PL=0
MOVL C01260 V=800.0 PL=0
MOVL C01261 V=800.0 PL=0
MOVL C01262 V=800.0 PL=0
MOVL C01263 V=800.0 PL=0
MOVL C01264 V=800.0 PL=0
MOVL C01265 V=800.0 PL=0
MOVL C01266 V=800.0 PL=0
MOVL C01267 V=800.0 PL=0
MOVL C01268 V=800.0 PL=0
MOVL C01269 V=800.0 PL=0
MOVL C01270 V=800.0 PL=0
MOVL C01271 V=800.0 PL=0
MOVL C01272 V=800.0 PL=0
MOVL C01273 V=800.0 PL=0
MOVL C01274 V=800.0 PL=0
MOVL C01275 V=800.0 PL=0
MOVL C01276 V=800.0 PL=0
MOVL C01277 V=800.0 PL=0
MOVL C01278 V=800.0 PL=0
MOVL C01279 V=800.0 PL=0
MOVL C01280 V=800.0 PL=0
MOVL C01281 V=800.0 PL=0
MOVL C01282 V=800.0 PL=0
MOVL C01283 V=800.0 PL=0
MOVL C01284 V=800.0 PL=0
MOVL C01285 V=800.0 PL=0
MOVL C01286 V=800.0 PL=0
MOVL C01287 V=800.0 PL=0
MOVL C01288 V=800.0 PL=0
MOVL C01289 V=800.0 PL=0
MOVL C01290 V=800.0 PL=0
MOVL C01291 V=800.0 PL=0
MOVL C01292 V=800.0 PL=0
MOVL C01293 V=800.0 PL=0
MOVL C01294 V=800.0 PL=0
MOVL C01295 V=800.0 PL=0
MOVL C01296 V=800.0 PL=0
MOVL C01297 V=800.0 PL=0
MOVL C01298 V=800.0 PL=0
MOVL C01299 V=800.0 PL=0
MOVL C01300 V=800.0 PL=0
MOVL C01301 V=800.0 PL=0
MOVL C01302 V=800.0 PL=0
MOVL C01303 V=800.0 PL=0
MOVL C01304 V=800.0 PL=0
MOVL C01305 V=800.0 PL=0
MOVL C01306 V=800.0 PL=0
MOVL C01307 V=800.0 PL=0
MOVL C01308 V=800.0 PL=0
MOVL C01309 V=800.0 PL=0
MOVL C01310 V=800.0 PL=0
MOVL C01311 V=800.0 PL=0
MOVL C01312 V=800.0 PL=0
MOVL C01313 V=800.0 PL=0
MOVL C01314 V=800.0 PL=0
MOVL C01315 V=800.0 PL=0
MOVL C01316 V=800.0 PL=0
MOVL C01317 V=800.0 PL=0
MOVL C01318 V=800.0 PL=0
MOVL C01319 V=800.0 PL=0
MOVL C01320 V=800.0 PL=0
MOVL C01321 V=800.0 PL=0
MOVL C01322 V=800.0 PL=0
MOVL C01323 V=800.0 PL=0
MOVL C01324 V=800.0 PL=0
MOVL C01325 V=800.0 PL=0
MOVL C01326 V=800.0 PL=0
MOVL C01327 V=800.0 PL=0
MOVL C01328 V=800.0 PL=0
MOVL C01329 V=800.0 PL=0
MOVL C01330 V=800.0 PL=0
MOVL C01331 V=800.0 PL=0
MOVL C01332 V=800.0 PL=0
MOVL C01333 V=800.0 PL=0
MOVL C01334 V=800.0 PL=0
MOVL C01335 V=800.0 PL=0
MOVL C01336 V=800.0 PL=0
MOVL C01337 V=800.0 PL=0
MOVL C01338 V=800.0 PL=0
MOVL C01339 V=800.0 PL=0
MOVL C01340 V=800.0 PL=0
MOVL C01341 V=800.0 PL=0
MOVL C01342 V=800.0 PL=0
MOVL C01343 V=800.0 PL=0
MOVL C01344 V=800.0 PL=0
MOVL C01345 V=800.0 PL=0
MOVL C01346 V=800.0 PL=0
MOVL C01347 V=800.0 PL=0
MOVL C01348 V=800.0 PL=0
MOVL C01349 V=800.0 PL=0
MOVL C01350 V=800.0 PL=0
MOVL C01351 V=800.0 PL=0
MOVL C01352 V=800.0 PL=0
MOVL C01353 V=800.0 PL=0
MOVL C01354 V=800.0 PL=0
MOVL C01355 V=800.0 PL=0
MOVL C01356 V=800.0 PL=0
MOVL C01357 V=800.0 PL=0
MOVL C01358 V=800.0 PL=0
MOVL C01359 V=800.0 PL=0
MOVL C01360 V=800.0 PL=0
MOVL C01361 V=800.0 PL=0
MOVL C01362 V=800.0 PL=0
MOVL C01363 V=800.0 PL=0
MOVL C01364 V=800.0 PL=0
MOVL C01365 V=800.0 PL=0
MOVL C01366 V=800.0 PL=0
MOVL C01367 V=800.0 PL=0
MOVL C01368 V=800.0 PL=0
MOVL C01369 V=800.0 PL=0
MOVL C01370 V=800.0 PL=0
MOVL C01371 V=800.0 PL=0
MOVL C01372 V=800.0 PL=0
MOVL C01373 V=800.0 PL=0
MOVL C01374 V=800.0 PL=0
MOVL C01375 V=800.0 PL=0
MOVL C01376 V=800.0 PL=0
MOVL C01377 V=800.0 PL=0
MOVL C01378 V=800.0 PL=0
MOVL C01379 V=800.0 PL=0
MOVL C01380 V=800.0 PL=0
MOVL C01381 V=800.0 PL=0
MOVL C01382 V=800.0 PL=0
MOVL C01383 V=800.0 PL=0
MOVL C01384 V=800.0 PL=0
MOVL C01385 V=800.0 PL=0
MOVL C01386 V=800.0 PL=0
MOVL C01387 V=800.0 PL=0
MOVL C01388 V=800.0 PL=0
MOVL C01389 V=800.0 PL=0
MOVL C01390 V=800.0 PL=0
MOVL C01391 V=800.0 PL=0
MOVL C01392 V=800.0 PL=0
MOVL C01393 V=800.0 PL=0
MOVL C01394 V=800.0 PL=0
MOVL C01395 V=800.0 PL=0
MOVL C01396 V=800.0 PL=0
MOVL C01397 V=800.0 PL=0
MOVL C01398 V=800.0 PL=0
MOVL C01399 V=800.0 PL=0
MOVL C01400 V=800.0 PL=0
MOVL C01401 V=800.0 PL=0
MOVL C01402 V=800.0 PL=0
MOVL C01403 V=800.0 PL=0
MOVL C01404 V=800.0 PL=0
MOVL C01405 V=800.0 PL=0
MOVL C01406 V=800.0 PL=0
MOVL C01407 V=800.0 PL=0
MOVL C01408 V=800.0 PL=0
MOVL C01409 V=800.0 PL=0
MOVL C01410 V=800.0 PL=0
MOVL C01411 V=800.0 PL=0
MOVL C01412 V=800.0 PL=0
MOVL C01413 V=800.0 PL=0
MOVL C01414 V=800.0 PL=0
MOVL C01415 V=800.0 PL=0
MOVL C01416 V=800.0 PL=0
MOVL C01417 V=800.0 PL=0
MOVL C01418 V=800.0 PL=0
MOVL C01419 V=800.0 PL=0
MOVL C01420 V=800.0 PL=0
MOVL C01421 V=800.0 PL=0
MOVL C01422 V=800.0 PL=0
MOVL C01423 V=800.0 PL=0
MOVL C01424 V=800.0 PL=0
MOVL C01425 V=800.0 PL=0
MOVL C01426 V=800.0 PL=0
MOVL C01427 V=800.0 PL=0
MOVL C01428 V=800.0 PL=0
MOVL C01429 V=800.0 PL=0
MOVL C01430 V=800.0 PL=0
MOVL C01431 V=800.0 PL=0
MOVL C01432 V=800.0 PL=0
MOVL C01433 V=800.0 PL=0
MOVL C01434 V=800.0 PL=0
MOVL C01435 V=800.0 PL=0
MOVL C01436 V=800.0 PL=0
MOVL C01437 V=800.0 PL=0
MOVL C01438 V=800.0 PL=0
MOVL C01439 V=800.0 PL=0
MOVL C01440 V=800.0 PL=0
MOVL C01441 V=800.0 PL=0
MOVL C01442 V=800.0 PL=0
MOVL C01443 V=800.0 PL=0
MOVL C01444 V=800.0 PL=0
MOVL C01445 V=800.0 PL=0
MOVL C01446 V=800.0 PL=0
MOVL C01447 V=800.0 PL=0
MOVL C01448 V=800.0 PL=0
MOVL C01449 V=800.0 PL=0
MOVL C01450 V=800.0 PL=0
MOVL C01451 V=800.0 PL=0
MOVL C01452 V=800.0 PL=0
MOVL C01453 V=800.0 PL=0
MOVL C01454 V=800.0 PL=0
MOVL C01455 V=800.0 PL=0
MOVL C01456 V=800.0 PL=0
MOVL C01457 V=800.0 PL=0
MOVL C01458 V=800.0 PL=0
MOVL C01459 V=800.0 PL=0
MOVL C01460 V=800.0 PL=0
MOVL C01461 V=800.0 PL=0
MOVL C01462 V=800.0 PL=0
MOVL C01463 V=800.0 PL=0
MOVL C01464 V=800.0 PL=0
MOVL C01465 V=800.0 PL=0
MOVL C01466 V=800.0 PL=0
MOVL C01467 V=800.0 PL=0
MOVL C01468 V=800.0 PL=0
MOVL C01469 V=800.0 PL=0
MOVL C01470 V=800.0 PL=0
MOVL C01471 V=800.0 PL=0
MOVL C01472 V=800.0 PL=0
MOVL C01473 V=800.0 PL=0
MOVL C01474 V=800.0 PL=0
MOVL C01475 V=800.0 PL=0
MOVL C01476 V=800.0 PL=0
MOVL C01477 V=800.0 PL=0
MOVL C01478 V=800.0 PL=0
MOVL C01479 V=800.0 PL=0
MOVL C01480 V=800.0 PL=0
MOVL C01481 V=800.0 PL=0
MOVL C01482 V=800.0 PL=0
MOVL C01483 V=800.0 PL=0
MOVL C01484 V=800.0 PL=0
MOVL C01485 V=800.0 PL=0
MOVL C01486 V=800.0 PL=0
MOVL C01487 V=800.0 PL=0
MOVL C01488 V=800.0 PL=0
MOVL C01489 V=800.0 PL=0
MOVL C01490 V=800.0 PL=0
MOVL C01491 V=800.0 PL=0
MOVL C01492 V=800.0 PL=0
MOVL C01493 V=800.0 PL=0
MOVL C01494 V=800.0 PL=0
MOVL C01495 V=800.0 PL=0
MOVL C01496 V=800.0 PL=0
MOVL C01497 V=800.0 PL=0
MOVL C01498 V=800.0 PL=0
MOVL C01499 V=800.0 PL=0
MOVL C01500 V=800.0 PL=0
MOVL C01501 V=800.0 PL=0
MOVL C01502 V=800.0 PL=0
MOVL C01503 V=800.0 PL=0
MOVL C01504 V=800.0 PL=0
MOVL C01505 V=800.0 PL=0
MOVL C01506 V=800.0 PL=0
MOVL C01507 V=800.0 PL=0
MOVL C01508 V=800.0 PL=0
MOVL C01509 V=800.0 PL=0
MOVL C01510 V=800.0 PL=0
MOVL C01511 V=800.0 PL=0
MOVL C01512 V=800.0 PL=0
MOVL C01513 V=800.0 PL=0
MOVL C01514 V=800.0 PL=0
MOVL C01515 V=800.0 PL=0
MOVL C01516 V=800.0 PL=0
MOVL C01517 V=800.0 PL=0
MOVL C01518 V=800.0 PL=0
MOVL C01519 V=800.0 PL=0
MOVL C01520 V=800.0 PL=0
MOVL C01521 V=800.0 PL=0
MOVL C01522 V=800.0 PL=0
MOVL C01523 V=800.0 PL=0
MOVL C01524 V=800.0 PL=0
MOVL C01525 V=800.0 PL=0
MOVL C01526 V=800.0 PL=0
MOVL C01527 V=800.0 PL=0
MOVL C01528 V=800.0 PL=0
MOVL C01529 V=800.0 PL=0
MOVL C01530 V=800.0 PL=0
MOVL C01531 V=800.0 PL=0
MOVL C01532 V=800.0 PL=0
MOVL C01533 V=800.0 PL=0
MOVL C01534 V=800.0 PL=0
MOVL C01535 V=800.0 PL=0
MOVL C01536 V=800.0 PL=0
MOVL C01537 V=800.0 PL=0
MOVL C01538 V=800.0 PL=0
MOVL C01539 V=800.0 PL=0
MOVL C01540 V=800.0 PL=0
MOVL C01541 V=800.0 PL=0
MOVL C01542 V=800.0 PL=0
MOVL C01543 V=800.0 PL=0
MOVL C01544 V=800.0 PL=0
MOVL C01545 V=800.0 PL=0
MOVL C01546 V=800.0 PL=0
MOVL C01547 V=800.0 PL=0
MOVL C01548 V=800.0 PL=0
MOVL C01549 V=800.0 PL=0
MOVL C01550 V=800.0 PL=0
MOVL C01551 V=800.0 PL=0
MOVL C01552 V=800.0 PL=0
MOVL C01553 V=800.0 PL=0
MOVL C01554 V=800.0 PL=0
MOVL C01555 V=800.0 PL=0
MOVL C01556 V=800.0 PL=0
MOVL C01557 V=800.0 PL=0
MOVL C01558 V=800.0 PL=0
MOVL C01559 V=800.0 PL=0
MOVL C01560 V=800.0 PL=0
MOVL C01561 V=800.0 PL=0
MOVL C01562 V=800.0 PL=0
MOVL C01563 V=800.0 PL=0
MOVL C01564 V=800.0 PL=0
MOVL C01565 V=800.0 PL=0
MOVL C01566 V=800.0 PL=0
MOVL C01567 V=800.0 PL=0
MOVL C01568 V=800.0 PL=0
MOVL C01569 V=800.0 PL=0
MOVL C01570 V=800.0 PL=0
MOVL C01571 V=800.0 PL=0
MOVL C01572 V=800.0 PL=0
MOVL C01573 V=800.0 PL=0
MOVL C01574 V=800.0 PL=0
MOVL C01575 V=800.0 PL=0
MOVL C01576 V=800.0 PL=0
MOVL C01577 V=800.0 PL=0
MOVL C01578 V=800.0 PL=0
MOVL C01579 V=800.0 PL=0
MOVL C01580 V=800.0 PL=0
MOVL C01581 V=800.0 PL=0
MOVL C01582 V=800.0 PL=0
MOVL C01583 V=800.0 PL=0
MOVL C01584 V=800.0 PL=0
MOVL C01585 V=800.0 PL=0
MOVL C01586 V=800.0 PL=0
MOVL C01587 V=800.0 PL=0
MOVL C01588 V=800.0 PL=0
MOVL C01589 V=800.0 PL=0
MOVL C01590 V=800.0 PL=0
MOVL C01591 V=800.0 PL=0
MOVL C01592 V=800.0 PL=0
MOVL C01593 V=800.0 PL=0
MOVL C01594 V=800.0 PL=0
MOVL C01595 V=800.0 PL=0
MOVL C01596 V=800.0 PL=0
MOVL C01597 V=800.0 PL=0
MOVL C01598 V=800.0 PL=0
MOVL C01599 V=800.0 PL=0
MOVL C01600 V=800.0 PL=0
MOVL C01601 V=800.0 PL=0
MOVL C01602 V=800.0 PL=0
MOVL C01603 V=800.0 PL=0
MOVL C01604 V=800.0 PL=0
MOVL C01605 V=800.0 PL=0
MOVL C01606 V=800.0 PL=0
MOVL C01607 V=800.0 PL=0
MOVL C01608 V=800.0 PL=0
MOVL C01609 V=800.0 PL=0
MOVL C01610 V=800.0 PL=0
MOVL C01611 V=800.0 PL=0
MOVL C01612 V=800.0 PL=0
MOVL C01613 V=800.0 PL=0
MOVL C01614 V=800.0 PL=0
MOVL C01615 V=800.0 PL=0
MOVL C01616 V=800.0 PL=0
MOVL C01617 V=800.0 PL=0
MOVL C01618 V=800.0 PL=0
MOVL C01619 V=800.0 PL=0
MOVL C01620 V=800.0 PL=0
MOVL C01621 V=800.0 PL=0
MOVL C01622 V=800.0 PL=0
MOVL C01623 V=800.0 PL=0
MOVL C01624 V=800.0 PL=0
MOVL C01625 V=800.0 PL=0
MOVL C01626 V=800.0 PL=0
MOVL C01627 V=800.0 PL=0
MOVL C01628 V=800.0 PL=0
MOVL C01629 V=800.0 PL=0
MOVL C01630 V=800.0 PL=0
MOVL C01631 V=800.0 PL=0
MOVL C01632 V=800.0 PL=0
MOVL C01633 V=800.0 PL=0
MOVL C01634 V=800.0 PL=0
MOVL C01635 V=800.0 PL=0
MOVL C01636 V=800.0 PL=0
MOVL C01637 V=800.0 PL=0
MOVL C01638 V=800.0 PL=0
MOVL C01639 V=800.0 PL=0
MOVL C01640 V=800.0 PL=0
MOVL C01641 V=800.0 PL=0
MOVL C01642 V=800.0 PL=0
MOVL C01643 V=800.0 PL=0
MOVL C01644 V=800.0 PL=0
MOVL C01645 V=800.0 PL=0
MOVL C01646 V=800.0 PL=0
MOVL C01647 V=800.0 PL=0
MOVL C01648 V=800.0 PL=0
MOVL C01649 V=800.0 PL=0
MOVL C01650 V=800.0 PL=0
MOVL C01651 V=800.0 PL=0
MOVL C01652 V=800.0 PL=0
MOVL C01653 V=800.0 PL=0
MOVL C01654 V=800.0 PL=0
MOVL C01655 V=800.0 PL=0
MOVL C01656 V=800.0 PL=0
MOVL C01657 V=800.0 PL=0
MOVL C01658 V=800.0 PL=0
MOVL C01659 V=800.0 PL=0
MOVL C01660 V=800.0 PL=0
MOVL C01661 V=800.0 PL=0
MOVL C01662 V=800.0 PL=0
MOVL C01663 V=800.0 PL=0
MOVL C01664 V=800.0 PL=0
MOVL C01665 V=800.0 PL=0
MOVL C01666 V=800.0 PL=0
MOVL C01667 V=800.0 PL=0
MOVL C01668 V=800.0 PL=0
MOVL C01669 V=800.0 PL=0
MOVL C01670 V=800.0 PL=0
MOVL C01671 V=800.0 PL=0
MOVL C01672 V=800.0 PL=0
MOVL C01673 V=800.0 PL=0
MOVL C01674 V=800.0 PL=0
MOVL C01675 V=800.0 PL=0
MOVL C01676 V=800.0 PL=0
MOVL C01677 V=800.0 PL=0
MOVL C01678 V=800.0 PL=0
MOVL C01679 V=800.0 PL=0
MOVL C01680 V=800.0 PL=0
MOVL C01681 V=800.0 PL=0
MOVL C01682 V=800.0 PL=0
MOVL C01683 V=800.0 PL=0
MOVL C01684 V=800.0 PL=0
MOVL C01685 V=800.0 PL=0
MOVL C01686 V=800.0 PL=0
MOVL C01687 V=800.0 PL=0
MOVL C01688 V=800.0 PL=0
MOVL C01689 V=800.0 PL=0
MOVL C01690 V=800.0 PL=0
MOVL C01691 V=800.0 PL=0
MOVL C01692 V=800.0 PL=0
MOVL C01693 V=800.0 PL=0
MOVL C01694 V=800.0 PL=0
MOVL C01695 V=800.0 PL=0
MOVL C01696 V=800.0 PL=0
MOVL C01697 V=800.0 PL=0
MOVL C01698 V=800.0 PL=0
MOVL C01699 V=800.0 PL=0
MOVL C01700 V=800.0 PL=0
MOVL C01701 V=800.0 PL=0
MOVL C01702 V=800.0 PL=0
MOVL C01703 V=800.0 PL=0
MOVL C01704 V=800.0 PL=0
MOVL C01705 V=800.0 PL=0
MOVL C01706 V=800.0 PL=0
MOVL C01707 V=800.0 PL=0
MOVL C01708 V=800.0 PL=0
MOVL C01709 V=800.0 PL=0
MOVL C01710 V=800.0 PL=0
MOVL C01711 V=800.0 PL=0
MOVL C01712 V=800.0 PL=0
MOVL C01713 V=800.0 PL=0
MOVL C01714 V=800.0 PL=0
MOVL C01715 V=800.0 PL=0
MOVL C01716 V=800.0 PL=0
MOVL C01717 V=800.0 PL=0
MOVL C01718 V=800.0 PL=0
MOVL C01719 V=800.0 PL=0
MOVL C01720 V=800.0 PL=0
MOVL C01721 V=800.0 PL=0
MOVL C01722 V=800.0 PL=0
MOVL C01723 V=800.0 PL=0
MOVL C01724 V=800.0 PL=0
MOVL C01725 V=800.0 PL=0
MOVL C01726 V=800.0 PL=0
MOVL C01727 V=800.0 PL=0
MOVL C01728 V=800.0 PL=0
MOVL C01729 V=800.0 PL=0
MOVL C01730 V=800.0 PL=0
MOVL C01731 V=800.0 PL=0
MOVL C01732 V=800.0 PL=0
MOVL C01733 V=800.0 PL=0
MOVL C01734 V=800.0 PL=0
MOVL C01735 V=800.0 PL=0
MOVL C01736 V=800.0 PL=0
MOVL C01737 V=800.0 PL=0
MOVL C01738 V=800.0 PL=0
MOVL C01739 V=800.0 PL=0
MOVL C01740 V=800.0 PL=0
MOVL C01741 V=800.0 PL=0
MOVL C01742 V=800.0 PL=0
MOVL C01743 V=800.0 PL=0
MOVL C01744 V=800.0 PL=0
MOVL C01745 V=800.0 PL=0
MOVL C01746 V=800.0 PL=0
MOVL C01747 V=800.0 PL=0
MOVL C01748 V=800.0 PL=0
MOVL C01749 V=800.0 PL=0
MOVL C01750 V=800.0 PL=0
MOVL C01751 V=800.0 PL=0
MOVL C01752 V=800.0 PL=0
MOVL C01753 V=800.0 PL=0
MOVL C01754 V=800.0 PL=0
MOVL C01755 V=800.0 PL=0
MOVL C01756 V=800.0 PL=0
MOVL C01757 V=800.0 PL=0
MOVL C01758 V=800.0 PL=0
MOVL C01759 V=800.0 PL=0
MOVL C01760 V=800.0 PL=0
MOVL C01761 V=800.0 PL=0
MOVL C01762 V=800.0 PL=0
MOVL C01763 V=800.0 PL=0
MOVL C01764 V=800.0 PL=0
MOVL C01765 V=800.0 PL=0
MOVL C01766 V=800.0 PL=0
MOVL C01767 V=800.0 PL=0
MOVL C01768 V=800.0 PL=0
MOVL C01769 V=800.0 PL=0
MOVL C01770 V=800.0 PL=0
MOVL C01771 V=800.0 PL=0
MOVL C01772 V=800.0 PL=0
MOVL C01773 V=800.0 PL=0
MOVL C01774 V=800.0 PL=0
MOVL C01775 V=800.0 PL=0
MOVL C01776 V=800.0 PL=0
MOVL C01777 V=800.0 PL=0
MOVL C01778 V=800.0 PL=0
MOVL C01779 V=800.0 PL=0
MOVL C01780 V=800.0 PL=0
MOVL C01781 V=800.0 PL=0
MOVL C01782 V=800.0 PL=0
MOVL C01783 V=800.0 PL=0
MOVL C01784 V=800.0 PL=0
MOVL C01785 V=800.0 PL=0
MOVL C01786 V=800.0 PL=0
MOVL C01787 V=800.0 PL=0
MOVL C01788 V=800.0 PL=0
MOVL C01789 V=800.0 PL=0
MOVL C01790 V=800.0 PL=0
MOVL C01791 V=800.0 PL=0
MOVL C01792 V=800.0 PL=0
MOVL C01793 V=800.0 PL=0
MOVL C01794 V=800.0 PL=0
MOVL C01795 V=800.0 PL=0
MOVL C01796 V=800.0 PL=0
MOVL C01797 V=800.0 PL=0
MOVL C01798 V=800.0 PL=0
MOVL C01799 V=800.0 PL=0
MOVL C01800 V=800.0 PL=0
MOVL C01801 V=800.0 PL=0
MOVL C01802 V=800.0 PL=0
MOVL C01803 V=800.0 PL=0
MOVL C01804 V=800.0 PL=0
MOVL C01805 V=800.0 PL=0
MOVL C01806 V=800.0 PL=0
MOVL C01807 V=800.0 PL=0
MOVL C01808 V=800.0 PL=0
MOVL C01809 V=800.0 PL=0
MOVL C01810 V=800.0 PL=0
MOVL C01811 V=800.0 PL=0
MOVL C01812 V=800.0 PL=0
MOVL C01813 V=800.0 PL=0
MOVL C01814 V=800.0 PL=0
MOVL C01815 V=800.0 PL=0
MOVL C01816 V=800.0 PL=0
MOVL C01817 V=800.0 PL=0
MOVL C01818 V=800.0 PL=0
MOVL C01819 V=800.0 PL=0
MOVL C01820 V=800.0 PL=0
MOVL C01821 V=800.0 PL=0
MOVL C01822 V=800.0 PL=0
MOVL C01823 V=800.0 PL=0
MOVL C01824 V=800.0 PL=0
MOVL C01825 V=800.0 PL=0
MOVL C01826 V=800.0 PL=0
MOVL C01827 V=800.0 PL=0
MOVL C01828 V=800.0 PL=0
MOVL C01829 V=800.0 PL=0
MOVL C01830 V=800.0 PL=0
MOVL C01831 V=800.0 PL=0
MOVL C01832 V=800.0 PL=0
MOVL C01833 V=800.0 PL=0
MOVL C01834 V=800.0 PL=0
MOVL C01835 V=800.0 PL=0
MOVL C01836 V=800.0 PL=0
MOVL C01837 V=800.0 PL=0
MOVL C01838 V=800.0 PL=0
MOVL C01839 V=800.0 PL=0
MOVL C01840 V=800.0 PL=0
MOVL C01841 V=800.0 PL=0
MOVL C01842 V=800.0 PL=0
MOVL C01843 V=800.0 PL=0
MOVL C01844 V=800.0 PL=0
MOVL C01845 V=800.0 PL=0
MOVL C01846 V=800.0 PL=0
MOVL C01847 V=800.0 PL=0
MOVL C01848 V=800.0 PL=0
MOVL C01849 V=800.0 PL=0
MOVL C01850 V=800.0 PL=0
MOVL C01851 V=800.0 PL=0
MOVL C01852 V=800.0 PL=0
MOVL C01853 V=800.0 PL=0
MOVL C01854 V=800.0 PL=0
MOVL C01855 V=800.0 PL=0
MOVL C01856 V=800.0 PL=0
MOVL C01857 V=800.0 PL=0
MOVL C01858 V=800.0 PL=0
MOVL C01859 V=800.0 PL=0
MOVL C01860 V=800.0 PL=0
MOVL C01861 V=800.0 PL=0
MOVL C01862 V=800.0 PL=0
MOVL C01863 V=800.0 PL=0
MOVL C01864 V=800.0 PL=0
MOVL C01865 V=800.0 PL=0
MOVL C01866 V=800.0 PL=0
MOVL C01867 V=800.0 PL=0
MOVL C01868 V=800.0 PL=0
MOVL C01869 V=800.0 PL=0
MOVL C01870 V=800.0 PL=0
MOVL C01871 V=800.0 PL=0
MOVL C01872 V=800.0 PL=0
MOVL C01873 V=800.0 PL=0
MOVL C01874 V=800.0 PL=0
MOVL C01875 V=800.0 PL=0
MOVL C01876 V=800.0 PL=0
MOVL C01877 V=800.0 PL=0
MOVL C01878 V=800.0 PL=0
MOVL C01879 V=800.0 PL=0
MOVL C01880 V=800.0 PL=0
MOVL C01881 V=800.0 PL=0
MOVL C01882 V=800.0 PL=0
MOVL C01883 V=800.0 PL=0
MOVL C01884 V=800.0 PL=0
MOVL C01885 V=800.0 PL=0
MOVL C01886 V=800.0 PL=0
MOVL C01887 V=800.0 PL=0
MOVL C01888 V=800.0 PL=0
MOVL C01889 V=800.0 PL=0
MOVL C01890 V=800.0 PL=0
MOVL C01891 V=800.0 PL=0
MOVL C01892 V=800.0 PL=0
MOVL C01893 V=800.0 PL=0
MOVL C01894 V=800.0 PL=0
MOVL C01895 V=800.0 PL=0
MOVL C01896 V=800.0 PL=0
MOVL C01897 V=800.0 PL=0
MOVL C01898 V=800.0 PL=0
MOVL C01899 V=800.0 PL=0
MOVL C01900 V=800.0 PL=0
MOVL C01901 V=800.0 PL=0
MOVL C01902 V=800.0 PL=0
MOVL C01903 V=800.0 PL=0
MOVL C01904 V=800.0 PL=0
MOVL C01905 V=800.0 PL=0
MOVL C01906 V=800.0 PL=0
MOVL C01907 V=800.0 PL=0
MOVL C01908 V=800.0 PL=0
MOVL C01909 V=800.0 PL=0
MOVL C01910 V=800.0 PL=0
MOVL C01911 V=800.0 PL=0
MOVL C01912 V=800.0 PL=0
MOVL C01913 V=800.0 PL=0
MOVL C01914 V=800.0 PL=0
MOVL C01915 V=800.0 PL=0
MOVL C01916 V=800.0 PL=0
MOVL C01917 V=800.0 PL=0
MOVL C01918 V=800.0 PL=0
MOVL C01919 V=800.0 PL=0
MOVL C01920 V=800.0 PL=0
MOVL C01921 V=800.0 PL=0
MOVL C01922 V=800.0 PL=0
MOVL C01923 V=800.0 PL=0
MOVL C01924 V=800.0 PL=0
MOVL C01925 V=800.0 PL=0
MOVL C01926 V=800.0 PL=0
MOVL C01927 V=800.0 PL=0
MOVL C01928 V=800.0 PL=0
MOVL C01929 V=800.0 PL=0
MOVL C01930 V=800.0 PL=0
MOVL C01931 V=800.0 PL=0
MOVL C01932 V=800.0 PL=0
MOVL C01933 V=800.0 PL=0
MOVL C01934 V=800.0 PL=0
MOVL C01935 V=800.0 PL=0
MOVL C01936 V=800.0 PL=0
MOVL C01937 V=800.0 PL=0
MOVL C01938 V=800.0 PL=0
MOVL C01939 V=800.0 PL=0
MOVL C01940 V=800.0 PL=0
MOVL C01941 V=800.0 PL=0
MOVL C01942 V=800.0 PL=0
MOVL C01943 V=800.0 PL=0
MOVL C01944 V=800.0 PL=0
MOVL C01945 V=800.0 PL=0
MOVL C01946 V=800.0 PL=0
MOVL C01947 V=800.0 PL=0
MOVL C01948 V=800.0 PL=0
MOVL C01949 V=800.0 PL=0
MOVL C01950 V=800.0 PL=0
MOVL C01951 V=800.0 PL=0
MOVL C01952 V=800.0 PL=0
MOVL C01953 V=800.0 PL=0
MOVL C01954 V=800.0 PL=0
MOVL C01955 V=800.0 PL=0
MOVL C01956 V=800.0 PL=0
MOVL C01957 V=800.0 PL=0
MOVL C01958 V=800.0 PL=0
MOVL C01959 V=800.0 PL=0
MOVL C01960 V=800.0 PL=0
MOVL C01961 V=800.0 PL=0
MOVL C01962 V=800.0 PL=0
MOVL C01963 V=800.0 PL=0
MOVL C01964 V=800.0 PL=0
MOVL C01965 V=800.0 PL=0
MOVL C01966 V=800.0 PL=0
MOVL C01967 V=800.0 PL=0
MOVL C01968 V=800.0 PL=0
MOVL C01969 V=800.0 PL=0
MOVL C01970 V=800.0 PL=0
MOVL C01971 V=800.0 PL=0
MOVL C01972 V=800.0 PL=0
MOVL C01973 V=800.0 PL=0
MOVL C01974 V=800.0 PL=0
MOVL C01975 V=800.0 PL=0
MOVL C01976 V=800.0 PL=0
MOVL C01977 V=800.0 PL=0
MOVL C01978 V=800.0 PL=0
MOVL C01979 V=800.0 PL=0
MOVL C01980 V=800.0 PL=0
MOVL C01981 V=800.0 PL=0
MOVL C01982 V=800.0 PL=0
MOVL C01983 V=800.0 PL=0
MOVL C01984 V=800.0 PL=0
MOVL C01985 V=800.0 PL=0
MOVL C01986 V=800.0 PL=0
MOVL C01987 V=800.0 PL=0
MOVL C01988 V=800.0 PL=0
MOVL C01989 V=800.0 PL=0
MOVL C01990 V=800.0 PL=0
MOVL C01991 V=800.0 PL=0
MOVL C01992 V=800.0 PL=0
MOVL C01993 V=800.0 PL=0
MOVL C01994 V=800.0 PL=0
MOVL C01995 V=800.0 PL=0
MOVL C01996 V=800.0 PL=0
MOVL C01997 V=800.0 PL=0
MOVL C01998 V=800.0 PL=0
MOVL C01999 V=800.0 PL=0
MOVL C02000 V=800.0 PL=0
MOVL C02001 V=800.0 PL=0
MOVL C02002 V=800.0 PL=0
MOVL C02003 V=800.0 PL=0
MOVL C02004 V=800.0 PL=0
MOVL C02005 V=800.0 PL=0
MOVL C02006 V=800.0 PL=0
MOVL C02007 V=800.0 PL=0
MOVL C02008 V=800.0 PL=0
MOVL C02009 V=800.0 PL=0
MOVL C02010 V=800.0 PL=0
MOVL C02011 V=800.0 PL=0
MOVL C02012 V=800.0 PL=0
MOVL C02013 V=800.0 PL=0
MOVL C02014 V=800.0 PL=0
MOVL C02015 V=800.0 PL=0
MOVL C02016 V=800.0 PL=0
MOVL C02017 V=800.0 PL=0
MOVL C02018 V=800.0 PL=0
MOVL C02019 V=800.0 PL=0
MOVL C02020 V=800.0 PL=0
MOVL C02021 V=800.0 PL=0
MOVL C02022 V=800.0 PL=0
MOVL C02023 V=800.0 PL=0
MOVL C02024 V=800.0 PL=0
MOVL C02025 V=800.0 PL=0
MOVL C02026 V=800.0 PL=0
MOVL C02027 V=800.0 PL=0
MOVL C02028 V=800.0 PL=0
MOVL C02029 V=800.0 PL=0
MOVL C02030 V=800.0 PL=0
MOVL C02031 V=800.0 PL=0
MOVL C02032 V=800.0 PL=0
MOVL C02033 V=800.0 PL=0
MOVL C02034 V=800.0 PL=0
MOVL C02035 V=800.0 PL=0
MOVL C02036 V=800.0 PL=0
MOVL C02037 V=800.0 PL=0
MOVL C02038 V=800.0 PL=0
MOVL C02039 V=800.0 PL=0
MOVL C02040 V=800.0 PL=0
MOVL C02041 V=800.0 PL=0
MOVL C02042 V=800.0 PL=0
MOVL C02043 V=800.0 PL=0
MOVL C02044 V=800.0 PL=0
MOVL C02045 V=800.0 PL=0
MOVL C02046 V=800.0 PL=0
MOVL C02047 V=800.0 PL=0
MOVL C02048 V=800.0 PL=0
MOVL C02049 V=800.0 PL=0
MOVL C02050 V=800.0 PL=0
MOVL C02051 V=800.0 PL=0
MOVL C02052 V=800.0 PL=0
MOVL C02053 V=800.0 PL=0
MOVL C02054 V=800.0 PL=0
MOVL C02055 V=800.0 PL=0
MOVL C02056 V=800.0 PL=0
MOVL C02057 V=800.0 PL=0
MOVL C02058 V=800.0 PL=0
MOVL C02059 V=800.0 PL=0
MOVL C02060 V=800.0 PL=0
MOVL C02061 V=800.0 PL=0
MOVL C02062 V=800.0 PL=0
MOVL C02063 V=800.0 PL=0
MOVL C02064 V=800.0 PL=0
MOVL C02065 V=800.0 PL=0
MOVL C02066 V=800.0 PL=0
MOVL C02067 V=800.0 PL=0
MOVL C02068 V=800.0 PL=0
MOVL C02069 V=800.0 PL=0
MOVL C02070 V=800.0 PL=0
MOVL C02071 V=800.0 PL=0
MOVL C02072 V=800.0 PL=0
MOVL C02073 V=800.0 PL=0
MOVL C02074 V=800.0 PL=0
MOVL C02075 V=800.0 PL=0
MOVL C02076 V=800.0 PL=0
MOVL C02077 V=800.0 PL=0
MOVL C02078 V=800.0 PL=0
MOVL C02079 V=800.0 PL=0
MOVL C02080 V=800.0 PL=0
MOVL C02081 V=800.0 PL=0
MOVL C02082 V=800.0 PL=0
MOVL C02083 V=800.0 PL=0
MOVL C02084 V=800.0 PL=0
MOVL C02085 V=800.0 PL=0
MOVL C02086 V=800.0 PL=0
MOVL C02087 V=800.0 PL=0
MOVL C02088 V=800.0 PL=0
MOVL C02089 V=800.0 PL=0
MOVL C02090 V=800.0 PL=0
MOVL C02091 V=800.0 PL=0
MOVL C02092 V=800.0 PL=0
MOVL C02093 V=800.0 PL=0
MOVL C02094 V=800.0 PL=0
MOVL C02095 V=800.0 PL=0
MOVL C02096 V=800.0 PL=0
MOVL C02097 V=800.0 PL=0
MOVL C02098 V=800.0 PL=0
MOVL C02099 V=800.0 PL=0
MOVL C02100 V=800.0 PL=0
MOVL C02101 V=800.0 PL=0
MOVL C02102 V=800.0 PL=0
MOVL C02103 V=800.0 PL=0
MOVL C02104 V=800.0 PL=0
MOVL C02105 V=800.0 PL=0
MOVL C02106 V=800.0 PL=0
MOVL C02107 V=800.0 PL=0
MOVL C02108 V=800.0 PL=0
MOVL C02109 V=800.0 PL=0
MOVL C02110 V=800.0 PL=0
MOVL C02111 V=800.0 PL=0
MOVL C02112 V=800.0 PL=0
MOVL C02113 V=800.0 PL=0
MOVL C02114 V=800.0 PL=0
MOVL C02115 V=800.0 PL=0
MOVL C02116 V=800.0 PL=0
MOVL C02117 V=800.0 PL=0
MOVL C02118 V=800.0 PL=0
MOVL C02119 V=800.0 PL=0
MOVL C02120 V=800.0 PL=0
MOVL C02121 V=800.0 PL=0
MOVL C02122 V=800.0 PL=0
MOVL C02123 V=800.0 PL=0
MOVL C02124 V=800.0 PL=0
MOVL C02125 V=800.0 PL=0
MOVL C02126 V=800.0 PL=0
MOVL C02127 V=800.0 PL=0
MOVL C02128 V=800.0 PL=0
MOVL C02129 V=800.0 PL=0
MOVL C02130 V=800.0 PL=0
MOVL C02131 V=800.0 PL=0
MOVL C02132 V=800.0 PL=0
MOVL C02133 V=800.0 PL=0
MOVL C02134 V=800.0 PL=0
MOVL C02135 V=800.0 PL=0
MOVL C02136 V=800.0 PL=0
MOVL C02137 V=800.0 PL=0
MOVL C02138 V=800.0 PL=0
MOVL C02139 V=800.0 PL=0
MOVL C02140 V=800.0 PL=0
MOVL C02141 V=800.0 PL=0
MOVL C02142 V=800.0 PL=0
MOVL C02143 V=800.0 PL=0
MOVL C02144 V=800.0 PL=0
MOVL C02145 V=800.0 PL=0
MOVL C02146 V=800.0 PL=0
MOVL C02147 V=800.0 PL=0
MOVL C02148 V=800.0 PL=0
MOVL C02149 V=800.0 PL=0
MOVL C02150 V=800.0 PL=0
MOVL C02151 V=800.0 PL=0
MOVL C02152 V=800.0 PL=0
